(* Logix 5000 project; controller CLASE_1 Emulate 5570 rev 28.11; software revision 28.02; part 11 of 15 *)
(* tags used below, declared in another part *)
   Cfg_FailOpen : BOOL;   // 1=Fail Open (energize to close), 0=Fail Closed (energize to open)
   PCmd_Open : BOOL;   // Program Command to Open Valve
   PCmd_Close : BOOL;   // Program Command to Close Valve
   OCmd_Open : BOOL;   // Operator Command to Open Valve
   OCmd_Close : BOOL;   // Operator Command to Close Valve
   Out : BOOL;   // 1=Energize Valve Solenoid
   P_ValveSO : BOOL;   // Unique Parameter Name for auto - discovery
   Wrk_Open : BOOL;   // 1=Requested to OPEN Valve, 0=Requested to CLOSE Valve
   Wrk_SimOpenT : TIMER;   // Simulation Delay until Opened
   Wrk_SimCloseT : TIMER;   // Simulation Delay until Closed
   Wrk_TransitStallT : TIMER;   // Timer for Transit Stall Check
   Wrk_FullStallT : TIMER;   // Timer for Full Stall Check
   Wrk_SimOpenLS : BOOL;   // Simulated valve Open Limit Switch
   Wrk_SimClosedLS : BOOL;   // Simulated valve Closed Limit Switch
(* P_ValveSO, continued *)

ROUTINE Prescan   (* ladder *)
// Clear Ownership, set to De-Energized state, clear "lurking" Commands
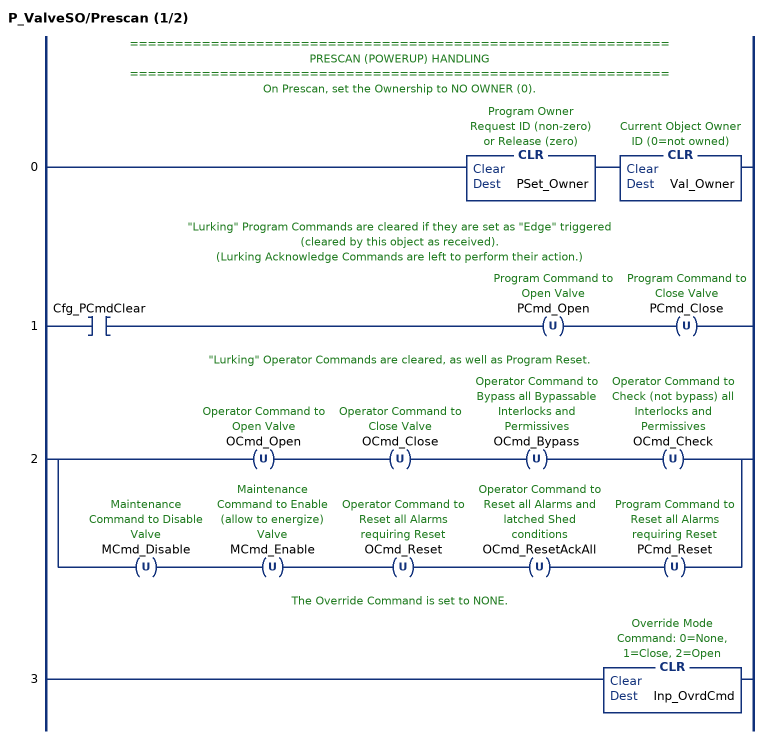
   // ============================================================
   // PRESCAN (POWERUP) HANDLING
   // ============================================================
   // On Prescan, set the Ownership to NO OWNER (0).
   0: CLR(PSet_Owner)CLR(Val_Owner);
   // "Lurking" Program Commands are cleared if they are set as "Edge" triggered
   // (cleared by this object as received).
   // (Lurking Acknowledge Commands are left to perform their action.)
   1: XIC(Cfg_PCmdClear)OTU(PCmd_Open)OTU(PCmd_Close);
   // "Lurking" Operator Commands are cleared, as well as Program Reset.
   2: [OTU(OCmd_Open) OTU(OCmd_Close) OTU(OCmd_Bypass) OTU(OCmd_Check) ,OTU(MCmd_Disable) OTU(MCmd_Enable) OTU(OCmd_Reset) OTU(OCmd_ResetAckAll) OTU(PCmd_Reset) ];
   // The Override Command is set to NONE.
   3: CLR(Inp_OvrdCmd);
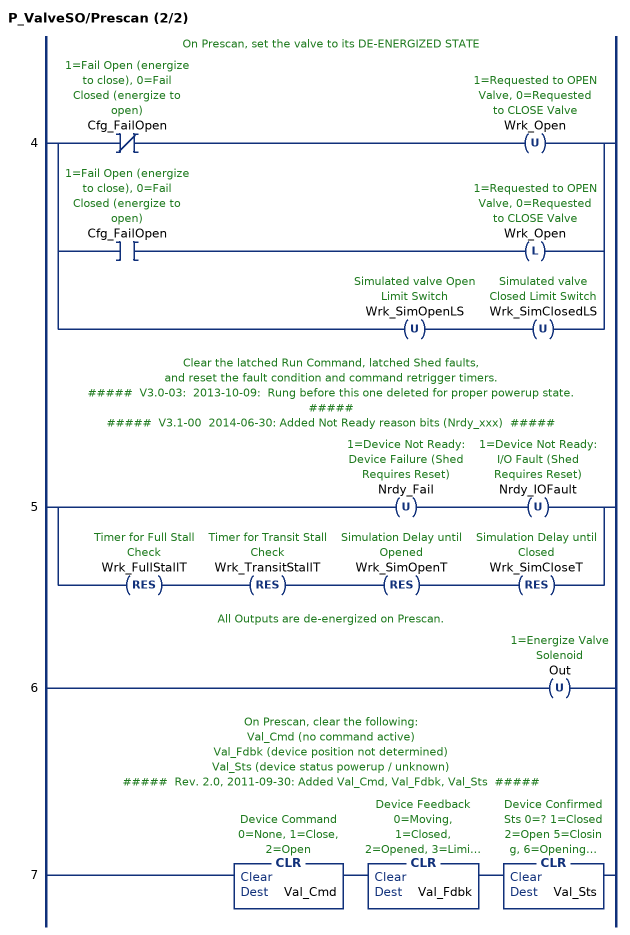
   // On Prescan, set the valve to its DE-ENERGIZED STATE
   4: [XIO(Cfg_FailOpen) OTU(Wrk_Open) ,XIC(Cfg_FailOpen) OTL(Wrk_Open) ,OTU(Wrk_SimOpenLS) OTU(Wrk_SimClosedLS) ];
   // Clear the latched Run Command, latched Shed faults,
   // and reset the fault condition and command retrigger timers.
   // #####  V3.0-03:  2013-10-09:  Rung before this one deleted for proper powerup state.  #####
   // #####  V3.1-00  2014-06-30: Added Not Ready reason bits (Nrdy_xxx)  #####
   5: [OTU(Nrdy_Fail) OTU(Nrdy_IOFault) ,RES(Wrk_FullStallT) RES(Wrk_TransitStallT) RES(Wrk_SimOpenT) RES(Wrk_SimCloseT) ];
   // All Outputs are de-energized on Prescan.
   6: OTU(Out);
   // On Prescan, clear the following:
   // Val_Cmd (no command active)
   // Val_Fdbk (device position not determined)
   // Val_Sts (device status powerup / unknown)
   // #####  Rev. 2.0, 2011-09-30: Added Val_Cmd, Val_Fdbk, Val_Sts  #####
   7: CLR(Val_Cmd)CLR(Val_Fdbk)CLR(Val_Sts);
END_ROUTINE
END_ADD_ON_INSTRUCTION

ADD_ON_INSTRUCTION P_VSD   (* revision 3.5 09 Release, vendor Rockwell Automation, ExecutePrescan, ExecuteEnableInFalse *)
// Variable Speed Drive
// Revision note:
// See V3.5-xx Release Notes for details. Modified to correct indication of motor RUNNING status in HAND mode, regardless of interlock/stop conditions.
// Help:
// Copyright © Rockwell Automation, Inc.  All Rights Reserved.
// This Instruction controls and monitors a Variable-Speed (AC or DC) Drive
// and provides:
// *  Starting drive, stopping drive, jogging drive, setting speed reference and setting direction
// *  Monitoring of run feedback, display of actual drive status, including accel, decel, direction, speed
// *  Detection of Failure to Start, Failure to Stop, Drive Fault/Not Ready
// *  Monitoring of Permissive conditions to allow starting
// *  Monitoring of Interlock conditions to stop drive or prevent starting
// *  Simulation, providing feedback of a working drive while disabling outputs
// *  Monitoring of I/O communication faults
// *  Alarms for Fail to Start, Fail to Stop, Interlock Trip, Drive Fault/Not Ready, I/O Fault
// *  Operation in Hand, Maintenance, Override, Program and Operator Modes
// *  "Available" status for use by automation logic to know whether drive
//       can be controlled by other objects.
// Modes are provided by a P_Mode AOI instance.
// Alarms are provided by P_Alarm AOI instances.
// Modes of operation: Operator, Program, Override, Maintenance, Hand
VAR_IN_OUT
   Ref_FaultCodeList : P_DescList[1]; {required}   // Tag containing List of Fault Codes (DINT) and their Descriptions (STRING)
END_VAR
VAR_INPUT
   Inp_SpeedFdbk : REAL; {visible}   // Speed Feedbak in Drive Units (typ. 0-32767 = 0 to max freq.)
   Inp_LastFaultCode : DINT;   // Most recent drive fault code (enumeration)
   Inp_Datalink : REAL; {visible}   // Auxiliary Signal (datalink) Input in Drive (raw) Units
   Inp_Ready : BOOL := 1; {visible}   // 1=Drive is ready to run
   Inp_Running : BOOL; {visible}   // 1=Drive is Running (active)
   Inp_CommandDir : BOOL := 1; {visible}   // 1=Drive is commanded Forward, 0=Drive is commanded Reverse
   Inp_ActualDir : BOOL := 1; {visible}   // 1=Drive is running Forward, 0=Drive is running Reverse
   Inp_Accelerating : BOOL; {visible}   // 1=Drive is accelerating
   Inp_Decelerating : BOOL; {visible}   // 1=Drive is decelerating
   Inp_Alarm : BOOL; {visible}   // 1=Drive has an Alarm Condition (see drive display or manual)
   Inp_Faulted : BOOL; {visible}   // 1=Drive has Faulted (see drive display or manual)
   Inp_AtSpeed : BOOL; {visible}   // 1=Drive is at commanded speed
   Inp_FwdPermOK : BOOL := 1; {visible}   // 1=Permissives OK, drive can start Forward
   Inp_FwdNBPermOK : BOOL := 1; {visible}   // 1=Non-Bypassable Permissives OK, drive can start Forward
   Inp_RevPermOK : BOOL := 1; {visible}   // 1=Permissives OK, drive can start Reverse
   Inp_RevNBPermOK : BOOL := 1; {visible}   // 1=Non-Bypassable Permissives OK, motor can start Reverse
   Inp_IntlkOK : BOOL := 1; {visible}   // 1=Interlocks OK, drive can start/run
   Inp_NBIntlkOK : BOOL := 1; {visible}   // 1=Non-Bypassable Interlocks OK, drive can start/run
   Inp_IOFault : BOOL;   // Input Communication Status 0=OK, 1=fail
   Inp_Sim : BOOL;   // 1=Simulate working drive; 0=Start/Stop/ Monitor actual drive
   Inp_Hand : ALIAS FOR Mode.Inp_Hand; {visible}
   Inp_Ovrd : ALIAS FOR Mode.Inp_Ovrd; {visible}
   Inp_OvrdCmd : SINT; {visible}   // Override Mode Command: 0=None, 1=Stop, 2=Start Fwd 3=Start Rev
   Inp_OvrdSpeed : REAL;   // Value to set Speed Reference in Override Mode (SpeedRef EU)
   Inp_OvrdOutDatalink : REAL;   // Value to set Output Datalink in Override Mode (OutDatalink EU)
   Inp_Reset : BOOL; {visible}   // 1=Reset drive fault conditions and latched Alarms
   Cfg_HasReverse : BOOL;   // 1=Drive can be run reverse, 0=Forward only
   Cfg_HasJog : BOOL;   // 1=Drive Jog Command enabled/visible, 0=Drive Jog Command not allowed
   Cfg_AllowLocal : BOOL;   // 1=Allow Local Start/Stop without alarm, 0=Start/Stop from HMI/prog only
   Cfg_HasRunFdbk : BOOL;   // 1=Drive provides feedback signal on Inp_Running when running
   Cfg_UseRunFdbk : BOOL;   // 1=Drive run feedback should be used for failure checking
   Cfg_HasSpeedFdbk : BOOL;   // 1=Drive provides speed feedback on Inp_SpeedFdbk
   Cfg_UseSpeedFdbk : BOOL;   // 1=Drive speed determines running state, 0=state determined by drive Active input bit
   Cfg_HasInpDatalink : BOOL;   // 1=A signal is connected to Inp_Datalink
   Cfg_HasOutDatalink : BOOL;   // 1=A signal is connected to Out_Datalink
   Cfg_HasFwdPermObj : BOOL;   // 1=Tells HMI a P_Perm is connected to Inp_FwdPerm
   Cfg_HasRevPermObj : BOOL;   // 1=Tells HMI a P_Perm is connected to Inp_RevPerm
   Cfg_HasIntlkObj : BOOL;   // 1=Tells HMI a P_Intlk is connected to Inp_Intlk
   Cfg_HasResInhObj : BOOL;   // 1=Tells HMI a P_ResInh Restart Inhibit is connected
   Cfg_HasRunTimeObj : BOOL;   // 1=Tells HMI a P_RunTime is connected
   Cfg_SetTrack : BOOL := 1;   // 1=PSets track OSets in Oper, OSets track PSets in Prog, 0=no tracking
   Cfg_SetTrackOvrdHand : BOOL;   // 1=Prog/Oper Settings track Override/Hand speed reference
   Cfg_PCmdClear : ALIAS FOR Mode.Cfg_PCmdClear;
   Cfg_ProgDefault : ALIAS FOR Mode.Cfg_ProgDefault;
   Cfg_OperStopPrio : BOOL;   // 1=OCmd_Stop has priority, accepted any time, 0=OCmd_Stop only in Oper, Maint Mode.
   Cfg_OCmdResets : BOOL;   // 1=New Oper drive cmd. resets fault, 0=reset req'd to clear fault
   Cfg_OvrdPermIntlk : BOOL;   // 1=Override ignores Bypassable Perm/ Intlk; 0=always use Perm/Intlk
   Cfg_ShedOnFailToStart : BOOL := 1;   // 1=Stop Motor and Alarm on Fail to Start; 0=Alarm only on Fail to Start
   Cfg_ShedOnIOFault : BOOL := 1;   // 1=Stop Motor and Alarm on I/O Fault; 0=Alarm only on I/O Fault
   Cfg_SimScaleEU : BOOL;   // 1=In simulation, scale Speed Ref EU to Speed Fdbk EU
   Cfg_SimScaleRaw : BOOL;   // 1=In simulation, scale Speed Ref EU to raw, then raw to Speed Fdbk EU
   Cfg_HasFailToStartAlm : ALIAS FOR FailToStart.Cfg_Exists;   // 1=Fail to Start Alarm exists and will be checked
   Cfg_HasFailToStopAlm : ALIAS FOR FailToStop.Cfg_Exists;   // 1=Fail to Stop Alarm exists and will be checked
   Cfg_HasIntlkTripAlm : ALIAS FOR IntlkTrip.Cfg_Exists;   // 1=Interlock Trip Alarm exists and will be checked
   Cfg_HasDriveFaultAlm : ALIAS FOR DriveFault.Cfg_Exists;   // 1=Drive Fault alarm exists and will be checked
   Cfg_HasIOFaultAlm : ALIAS FOR IOFault.Cfg_Exists;   // 1=I/O Fault Alarm exists and will be checked
   Cfg_FailToStartResetReqd : ALIAS FOR FailToStart.Cfg_ResetReqd;   // 1=Reset requied to clear Fail to Start Alarm
   Cfg_FailToStopResetReqd : ALIAS FOR FailToStop.Cfg_ResetReqd;   // 1=Reset required to clear Fail to Stop Alarm
   Cfg_IntlkTripResetReqd : ALIAS FOR IntlkTrip.Cfg_ResetReqd;   // 1=Reset required to clear Interlock Trip Alarm
   Cfg_DriveFaultResetReqd : ALIAS FOR DriveFault.Cfg_ResetReqd;   // 1=Reset required to clear Drive Fault Alarm
   Cfg_IOFaultResetReqd : ALIAS FOR IOFault.Cfg_ResetReqd;   // 1=Reset required to clear I/O Fault Alarm
   Cfg_FailToStartAckReqd : ALIAS FOR FailToStart.Cfg_AckReqd;   // 1=Acknowledge required for Fail to Start Alarm
   Cfg_FailToStopAckReqd : ALIAS FOR FailToStop.Cfg_AckReqd;   // 1=Acknowledge required for Fail to Stop Alarm
   Cfg_IntlkTripAckReqd : ALIAS FOR IntlkTrip.Cfg_AckReqd;   // 1=Acknowledge required for Interlock Trip Alarm
   Cfg_DriveFaultAckReqd : ALIAS FOR DriveFault.Cfg_AckReqd;   // 1=Acknowledge required for Drive Fault Alarm
   Cfg_IOFaultAckReqd : ALIAS FOR IOFault.Cfg_AckReqd;   // 1=Acknowledge required for I/O Fault Alarm
   Cfg_FailToStartSeverity : ALIAS FOR FailToStart.Cfg_Severity;   // Fail To Start Alarm Severity: 1..250=Low, 251..500=Medium, 501..750=High, 751..1000=Urgent
   Cfg_FailToStopSeverity : ALIAS FOR FailToStop.Cfg_Severity;   // Fail To Stop Alarm Severity: 1..250=Low, 251..500=Medium, 501..750=High, 751..1000=Urgent
   Cfg_IntlkTripSeverity : ALIAS FOR IntlkTrip.Cfg_Severity;   // Interlock Trip Alarm Severity: 1..250=Low, 251..500=Medium, 501..750=High, 751..1000=Urgent
   Cfg_DriveFaultSeverity : ALIAS FOR DriveFault.Cfg_Severity;   // Drive Fault Alarm Severity: 1..250=Low, 251..500=Medium, 501..750=High, 751..1000=Urgent
   Cfg_IOFaultSeverity : ALIAS FOR IOFault.Cfg_Severity;   // I/O Fault Alarm Severity: 1..250=Low, 251..500=Medium, 501..750=High, 751..1000=Urgent
   Cfg_MinSpdRef : REAL;   // Minimum Speed Reference in EU (for limiting)
   Cfg_MaxSpdRef : REAL := 60.0;   // Maximum Speed Reference in EU (for limiting)
   Cfg_SpeedRefRawMin : REAL;   // Speed Reference Minimum in Drive (raw) Units (for scaling)
   Cfg_SpeedRefRawMax : REAL := 32767.0;   // Speed Reference Maximum in Drive (raw) Units (for scaling)
   Cfg_SpeedRefEUMin : REAL;   // Speed Reference Minimum in Engineering Units (for scaling)
   Cfg_SpeedRefEUMax : REAL := 130.0;   // Speed Reference Maximum in Engineering Units (for scaling)
   Cfg_SpeedFdbkRawMin : REAL;   // Speed Feedback Minimum in Drive (raw) Units (for scaling)
   Cfg_SpeedFdbkRawMax : REAL := 32767.0;   // Speed Feedback Maximum in Drive (raw) Units (for scaling)
   Cfg_SpeedFdbkEUMin : REAL;   // Speed Feedback Minimum in Engineering Units (for scaling)
   Cfg_SpeedFdbkEUMax : REAL := 130.0;   // Speed Feedback Maximum in Engineering Units (for scaling)
   Cfg_InpDatalinkRawMin : REAL;   // Input Datalink Minimum in Drive (raw) Units (for scaling)
   Cfg_InpDatalinkRawMax : REAL := 4095.0;   // Input Datalink Maximum in Drive (raw) Units (for scaling)
   Cfg_InpDatalinkEUMin : REAL;   // Input Datalink Minimum in Engineering Units (for scaling)
   Cfg_InpDatalinkEUMax : REAL := 409.5;   // Input Datalink Maximum in Engineering Units (for scaling)
   Cfg_OutDatalinkMin : REAL;   // Minimum Output Datalink in EU (for limiting)
   Cfg_OutDatalinkMax : REAL := 100.0;   // Maximum Output Datalink in EU (for limiting)
   Cfg_OutDatalinkRawMin : REAL;   // Output Datalink Minimum in Drive (raw) Units (for scaling)
   Cfg_OutDatalinkRawMax : REAL := 4095.0;   // Output Datalink Maximum in Drive (raw) Units (for scaling)
   Cfg_OutDatalinkEUMin : REAL;   // Output Datalink Minimum in Engineering Units (for scaling)
   Cfg_OutDatalinkEUMax : REAL := 409.5;   // Output Datalink Maximum in Engineering Units (for scaling)
   Cfg_SimRampT : DINT := 10;   // Time to ramp speed fdbk when in Simulation (sec)
   Cfg_FailToStartT : DINT := 15;   // Time after Start to get Run Feedback before Fault (sec)
   Cfg_FailToStopT : DINT := 15;   // Time after Stop to drop Run Feedback before Fault (sec)
   Cfg_ResetPulseT : DINT := 2;   // Time to pulse Out_Reset to clear drive fault
   Cfg_MaxJogT : REAL;   // Maximum jog time (sec, 0=unlimited)
   Cfg_OperKeep : SINT;   // Oper keeps control in Prog Mode: .0=Reference, .1=Start/Stop, .2=Fwd/Rev, .3=OutDatalink
   Cfg_ProgKeep : SINT;   // Prog keeps control in Oper Mode: .0=Reference, .1=Start/Stop, .2=Fwd/Rev, .3=OutDatalink
   PSet_SpeedRef : REAL;   // Program Setting of Speed Reference (EU)
   PSet_OutDatalink : REAL;   // Program Setting of Output Datalink (EU)
   PSet_Owner : DINT;   // Program Owner Request ID (non-zero) or Release (zero)
   OSet_SpeedRef : REAL;   // Operator Setting of Speed Reference (EU)
   OSet_OutDatalink : REAL;   // Operator Setting of Output Datalink (EU)
   PCmd_Start : BOOL;   // Program Command to Start Drive
   PCmd_Stop : BOOL;   // Program Command to Stop Drive
   PCmd_Fwd : BOOL;   // Program Command to set direction to Fowrard
   PCmd_Rev : BOOL;   // Program Command to set direction to Reverse
   PCmd_Acq : ALIAS FOR Mode.PCmd_Acq;
   PCmd_Rel : ALIAS FOR Mode.PCmd_Rel;
   PCmd_Lock : ALIAS FOR Mode.PCmd_Lock;
   PCmd_Unlock : ALIAS FOR Mode.PCmd_Unlock;
   PCmd_Reset : BOOL;   // Program Command to Reset drive fault and all Alarms requiring Reset
   PCmd_FailToStartAck : ALIAS FOR FailToStart.PCmd_Ack;   // Program Command to Acknowledge Fail to Start Alarm
   PCmd_FailToStartSuppress : ALIAS FOR FailToStart.PCmd_Suppress;   // Program Command to Suppress Fail to Start Alarm
   PCmd_FailToStartUnsuppress : ALIAS FOR FailToStart.PCmd_Unsuppress;   // Program Command to Unsuppress Fail to Start Alarm
   PCmd_FailToStartUnshelve : ALIAS FOR FailToStart.PCmd_Unshelve;   // Program Command to Unshelve Fail to Start Alarm
   PCmd_FailToStopAck : ALIAS FOR FailToStop.PCmd_Ack;   // Program Command to Acknowledge Fail to Stop Alarm
   PCmd_FailToStopSuppress : ALIAS FOR FailToStop.PCmd_Suppress;   // Program Command to Suppress Fail to Stop Alarm
   PCmd_FailToStopUnsuppress : ALIAS FOR FailToStop.PCmd_Unsuppress;   // Program Command to Unsuppress Fail to Stop Alarm
   PCmd_FailToStopUnshelve : ALIAS FOR FailToStop.PCmd_Unshelve;   // Program Command to Unshelve Fail to Stop Alarm
   PCmd_IntlkTripAck : ALIAS FOR IntlkTrip.PCmd_Ack;   // Program Command to Acknowledge Interlock Trip Alarm
   PCmd_IntlkTripSuppress : ALIAS FOR IntlkTrip.PCmd_Suppress;   // Program Command to Suppress Interlock Trip Alarm
   PCmd_IntlkTripUnsuppress : ALIAS FOR IntlkTrip.PCmd_Unsuppress;   // Program Command to Unsuppress Interlock Trip Alarm
   PCmd_IntlkTripUnshelve : ALIAS FOR IntlkTrip.PCmd_Unshelve;   // Program Command to Unshelve Interlock Trip Alarm
   PCmd_DriveFaultAck : ALIAS FOR DriveFault.PCmd_Ack;   // Program Command to Acknowledge Drive Fault Alarm
   PCmd_DriveFaultSuppress : ALIAS FOR DriveFault.PCmd_Suppress;   // Program Command to Suppress Drive Fault Alarm
   PCmd_DriveFaultUnsuppress : ALIAS FOR DriveFault.PCmd_Unsuppress;   // Program Command to Unsuppress Drive Fault Alarm
   PCmd_DriveFaultUnshelve : ALIAS FOR DriveFault.PCmd_Unshelve;   // Program Command to Unshelve Drive Fault Alarm
   PCmd_IOFaultAck : ALIAS FOR IOFault.PCmd_Ack;   // Program Command to Acknowledge I/O Fault Alarm
   PCmd_IOFaultSuppress : ALIAS FOR IOFault.PCmd_Suppress;   // Program Command to Suppress I/O Fault Alarm
   PCmd_IOFaultUnsuppress : ALIAS FOR IOFault.PCmd_Unsuppress;   // Program Command to Unsuppress I/O Fault Alarm
   PCmd_IOFaultUnshelve : ALIAS FOR IOFault.PCmd_Unshelve;   // Program Command to Unshelve I/O Fault Alarm
   OCmd_Start : BOOL;   // Operator Command to Start Drive
   OCmd_Stop : BOOL;   // Operator Command to Stop Drive
   OCmd_Jog : BOOL;   // Operator Command to Jog Drive (not cleared by P_VSD!)
   OCmd_Fwd : BOOL;   // Operator Command to set direction to Forward
   OCmd_Rev : BOOL;   // Operator Command to set direction to Reverse
   OCmd_Bypass : BOOL;   // Operator Command to Bypass all Bypassable Interlocks and Permissives
   OCmd_Check : BOOL;   // Operator Command to Check (not bypass) all Interlocks and Permissives
   MCmd_Disable : BOOL;   // Maintenance Command to Disable Drive
   MCmd_Enable : BOOL;   // Maintenance Command to Enable (allow to run) Drive
   MCmd_Acq : ALIAS FOR Mode.MCmd_Acq;
   MCmd_Rel : ALIAS FOR Mode.MCmd_Rel;
   OCmd_AcqLock : ALIAS FOR Mode.OCmd_AcqLock;
   OCmd_Unlock : ALIAS FOR Mode.OCmd_UnlockRel;
   OCmd_Reset : BOOL;   // Operator Command to Reset all Alarms requiring Reset
   OCmd_ResetAckAll : BOOL;   // Operator Command to Reset all Alarms and latched Shed conditions
END_VAR
VAR_OUTPUT
   Out_SpeedRef : REAL; {access Read Only, visible}   // Drive Speed Reference in Drive Units (typ. 0-32767 = 0 to max freq.)
   Out_Datalink : REAL; {access Read Only, visible}   // Auxiliary Signal (datalink) Output in Drive (raw) Units
   Out_Run : BOOL; {access Read Only}   // 1=Start/Run Drive, 0=Stop Drive (for held starter type)
   Out_Stop : BOOL; {access Read Only, visible}   // 1=Stop Drive, 0=drive left in current state
   Out_Start : BOOL; {access Read Only, visible}   // 1=Start Drive, 0=drive left in current state
   Out_Jog : BOOL; {access Read Only, visible}   // 1=Jog drive at Jog Speed, -->0=stop jogging
   Out_ClearFault : BOOL; {access Read Only, visible}   // 1=Attempt to clear Drive Fault
   Out_Fwd : BOOL; {access Read Only, visible}   // 1=Set drive direction to Forward
   Out_Rev : BOOL; {access Read Only, visible}   // 1=Set drive direction to Reverse
   Val_SpeedRef : REAL; {access Read Only, visible}   // Speed Reference (target) to drive
   Val_SpeedFdbk : REAL; {access Read Only, visible}   // Speed Feedback (actual) from drive
   Val_InpDatalink : REAL; {access Read Only, visible}   // Input Datalink value from drive
   Val_OutDatalink : REAL; {access Read Only, visible}   // Output Datalink value to drive
   Val_SpeedRefEUMin : REAL; {access Read Only}   // Minimum of Speed Reference = MIN (Cfg_SpeedFdbkEUMin, Cfg_SpeedFdbkEUMax)
   Val_SpeedRefEUMax : REAL := 130.0; {access Read Only}   // Maximum of Speed Reference = MAX (Cfg_SpeedFdbkEUMin, Cfg_SpeedFdbkEUMax)
   Val_SpeedFdbkEUMin : REAL; {access Read Only}   // Minimum of Speed Feedback = MIN (Cfg_SpeedFdbkEUMin, Cfg_SpeedFdbkEUMax)
   Val_SpeedFdbkEUMax : REAL := 130.0; {access Read Only}   // Maximum of Speed Feedback = MAX (Cfg_SpeedFdbkEUMin, Cfg_SpeedFdbkEUMax)
   Val_LastFaultCode : DINT; {access Read Only}   // Most recent drive fault code (enumeration)
   SrcQ_IO : SINT; {access Read Only}   // Source and Quality of primary I/O (enumeration)
   SrcQ : SINT; {access Read Only}   // Source and Quality of primary Val/Sts (enumeration)
   Val_Cmd : SINT; {access Read Only}   // Device Command 0=None, 1=Stop, 2=StartFwd 3=StartRev 4=JogFwd 5=JogRev
   Val_Fdbk : SINT; {access Read Only}   // Device Feedback 0=Stopped, 1=Running Fwd 2=Running Rev 3=Accelerating 4=Decelerating
   Val_Sts : SINT; {access Read Only}   // Device Confirmed Sts 0? 1=Stop 2=RunF 3=RunR 4=JogF 5=JogR 6=Stopping 7=Starting F 8=Starting R, 33=Disabled
   Val_Fault : SINT; {access Read Only, visible}   // Device Fault Status 0=None, 16=Fail to Start, 17 = Fail to Stop, 18=Drive Fault, 32=I/O Fault, 34=Config Error
   Val_Mode : ALIAS FOR Mode.Val; {access Read Only}
   Val_Owner : DINT; {access Read Only}   // Current Object Owner ID (0=not owned)
   Val_Notify : SINT; {access Read Only}   // Current Alarm Level and Acknowledgement (enumeration)
   Sts_Stopped : BOOL; {access Read Only, visible}   // 1=Drive requested to stop and is confirmed stopped
   Sts_Starting : BOOL; {access Read Only, visible}   // 1=Drive requested to run and awaiting run feedback
   Sts_Running : BOOL; {access Read Only, visible}   // 1=Drive requested to run and is confirmed running
   Sts_Stopping : BOOL; {access Read Only, visible}   // 1=Drive requested to stop and awaiting stopped feedback
   Sts_Jogging : BOOL; {access Read Only, visible}   // 1=Drive requested to Jog
   Sts_CommandDir : BOOL; {access Read Only}   // 1=Drive commanded to Forward, 0=Reverse
   Sts_ActualDir : BOOL; {access Read Only, visible}   // 1=Drive Actual direction is Forward, 0=Reverse
   Sts_Accel : BOOL; {access Read Only}   // 1=Drive is Accelerating
   Sts_Decel : BOOL; {access Read Only}   // 1=Drive is Decelerating
   Sts_NotReady : BOOL; {access Read Only}   // 1=Drive is Not Ready (cannot be started) Check alarms, stops, faults
   Sts_Alarm : BOOL; {access Read Only, visible}   // 1=Drive has an Alarm (see drive display or manual)
   Sts_AtSpeed : BOOL; {access Read Only, visible}   // 1=Drive is running at reference speed
   Sts_SpeedLimited : BOOL; {access Read Only, visible}   // 1=Speed Reference Setting exceeds configured Max/Min limit
   Sts_Available : BOOL; {access Read Only, visible}   // 1=Drive available for control by automation (Prog)
   Sts_Bypass : BOOL; {access Read Only}   // 1=Bypassable Interlocks and Permissives are Bypassed
   Sts_BypActive : BOOL; {access Read Only}   // 1=Bypassing Active (Bypassed or Maintenance)
   Sts_Disabled : BOOL; {access Read Only}   // 1=Drive is Disabled
   Sts_NotRdy : BOOL; {access Read Only}   // 1=Device Not Ready, see detail bits for reason
   Nrdy_Disabled : BOOL; {access Read Only}   // 1=Device Not Ready: Device Disabled by Maintenance
   Nrdy_CfgErr : BOOL; {access Read Only}   // 1=Device Not Ready: Configuration Error
   Nrdy_Intlk : BOOL; {access Read Only}   // 1=Device Not Ready: Interlock Not OK
   Nrdy_Perm : BOOL; {access Read Only}   // 1=Device Not Ready: Permissive Not OK
   Nrdy_OperPrio : BOOL; {access Read Only}   // 1=Device Not Ready: Operator State 0 Priority Command Requires Reset
   Nrdy_Fail : BOOL; {access Read Only}   // 1=Device Not Ready: Device Failure (Shed Requires Reset)
   Nrdy_IOFault : BOOL; {access Read Only}   // 1=Device Not Ready: I/O Fault (Shed Requires Reset)
   Nrdy_Trip : BOOL; {access Read Only}   // 1=Device not Ready: Deivce Tripped (Drive Fault)
   Nrdy_DriveNR : BOOL; {access Read Only}   // 1=Device Note Ready: Drive Not Ready
   Nrdy_NoMode : BOOL; {access Read Only}   // 1=Device Not Ready: Device Logic Disabled / NO Mode
   Sts_MaintByp : BOOL; {access Read Only}   // 1=A Maintenance Bypass is Active, display icon
   Sts_AlmInh : BOOL; {access Read Only}   // 1=An Alarm is Shelved, Disabled or Suppressed, display icon
   Sts_Err : BOOL; {access Read Only, visible}   // 1=Error in Config: see detail bits for reason
   Err_Timer : BOOL; {access Read Only}   // 1=Error in Config: Invalid Check or Reset Pulse Time (use 0 to 2147483)
   Err_Sim : BOOL; {access Read Only}   // 1=Error in Config: simulation timer preset: use 0 to 2147483)
   Err_Alarm : BOOL; {access Read Only}   // 1=Error in Config: Alarm Min On Time, Shelf Time, Severity
   Err_FdbkRaw : BOOL; {access Read Only}   // 1=Erron in Config: Speed Fdbk Raw Min = Max
   Err_FdbkEU : BOOL; {access Read Only}   // 1=Error in Config: Speed Fdbk EU Min = Max
   Err_RefLim : BOOL; {access Read Only}   // 1=Error in Config: Speed Ref Limit Min > Max
   Err_RefEU : BOOL; {access Read Only}   // 1=Error in Config: Speed Ref EU Min = Max
   Err_RefRaw : BOOL; {access Read Only}   // 1=Error in Config: Speed Ref Raw Min = Max
   Err_InpDLRaw : BOOL; {access Read Only}   // 1=Error in Config: Input Datalink Raw Min = Max
   Err_InpDLEU : BOOL; {access Read Only}   // 1=Error in Config: Input Datalink EU Min = Max
   Err_OutDLLim : BOOL; {access Read Only}   // 1=Error in Config: Output Datalink Limits Min > Max
   Err_OutDLEU : BOOL; {access Read Only}   // 1=Error in Config: Output Datalink EU Min = Max
   Err_OutDLRaw : BOOL; {access Read Only}   // 1=Error in Config: Output Datalink Raw Min = Max
   Sts_Hand : ALIAS FOR Mode.Sts_Hand; {access Read Only, visible}
   Sts_Maint : ALIAS FOR Mode.Sts_Maint; {access Read Only, visible}
   Sts_Ovrd : ALIAS FOR Mode.Sts_Ovrd; {access Read Only, visible}
   Sts_Prog : ALIAS FOR Mode.Sts_Prog; {access Read Only, visible}
   Sts_Oper : ALIAS FOR Mode.Sts_Oper; {access Read Only, visible}
   Sts_ProgOperLock : ALIAS FOR Mode.Sts_ProgOperLock; {access Read Only}
   Sts_NoMode : ALIAS FOR Mode.Sts_NoMode; {access Read Only}
   Sts_MAcqRcvd : ALIAS FOR Mode.Sts_MAcqRcvd; {access Read Only}
   Sts_FailToStart : ALIAS FOR FailToStart.Inp;   // 1=Drive Failed to Start (One-Shot)
   Alm_FailToStart : ALIAS FOR FailToStart.Alm;   // 1=Drive Fail to Start Alarm
   Ack_FailToStart : ALIAS FOR FailToStart.Ack;   // 1=Fail to Start Alarm has been acknowledged
   Sts_FailToStartDisabled : ALIAS FOR FailToStart.Disabled;   // 1=Fail to Start Alarm has been Disabled by Maintenance
   Sts_FailToStartShelved : ALIAS FOR FailToStart.Shelved;   // 1=Fail to Start Alarm has been Shelved by Operator
   Sts_FailToStartSuppressed : ALIAS FOR FailToStart.Suppressed;   // 1=Fail to Start Alarm has been Suppressed by Program
   Sts_FailToStop : ALIAS FOR FailToStop.Inp;   // 1=Drive Failed to Stop
   Alm_FailToStop : ALIAS FOR FailToStop.Alm;   // 1=Drive Fail to Stop Alarm
   Ack_FailToStop : ALIAS FOR FailToStop.Ack;   // 1=Fail to Stop Alarm has been acknowledged
   Sts_FailToStopDisabled : ALIAS FOR FailToStop.Disabled;   // 1=Fail to Stop Alarm has been Disabled by Maintenance
   Sts_FailToStopShelved : ALIAS FOR FailToStop.Shelved;   // 1=Fail to Stop Alarm has been Shelved by Operator
   Sts_FailToStopSuppressed : ALIAS FOR FailToStop.Suppressed;   // 1=Fail to Stop Alarm has been Suppressed by Program
   Sts_IntlkTrip : ALIAS FOR IntlkTrip.Inp;   // 1=Drive was stopped by an Interlock NOT OK (One-Shot)
   Alm_IntlkTrip : ALIAS FOR IntlkTrip.Alm;   // 1=Alarm: Drive stopped by an Interlock NOT OK
   Ack_IntlkTrip : ALIAS FOR IntlkTrip.Ack;   // 1=Interlock Trip Alarm has been acknowledged
   Sts_IntlkTripDisabled : ALIAS FOR IntlkTrip.Disabled;   // 1=Interlock Trip Alarm has been Disabled by Maintenance
   Sts_IntlkTripShelved : ALIAS FOR IntlkTrip.Shelved;   // 1=Interlock Trip Alarm has been Shelved by Operator
   Sts_IntlkTripSuppressed : ALIAS FOR IntlkTrip.Suppressed;   // 1=Interlock Trip Alarm has been Suppressed by Program
   Sts_DriveFault : ALIAS FOR DriveFault.Inp;   // 1=Drive Fault (see drive display or manual)
   Alm_DriveFault : ALIAS FOR DriveFault.Alm;   // 1=Alarm: Drive Fault (see drive display or manual)
   Ack_DriveFault : ALIAS FOR DriveFault.Ack;   // 1=Drive Fault Alarm has been acknowledged
   Sts_DriveFaultDisabled : ALIAS FOR DriveFault.Disabled;   // 1=Drive Fault Alarm has been Disabled by Maintenance
   Sts_DriveFaultShelved : ALIAS FOR DriveFault.Shelved;   // 1=Drive Fault Alarm has been Shelved by Operator
   Sts_DriveFaultSuppressed : ALIAS FOR DriveFault.Suppressed;   // 1=Drive Fault Alarm has been Suppressed by Program
   Sts_IOFault : ALIAS FOR IOFault.Inp;   // I/O Comm Fault Status (0=OK, 1=Bad)
   Alm_IOFault : ALIAS FOR IOFault.Alm;   // 1=I/O Fault Alarm
   Ack_IOFault : ALIAS FOR IOFault.Ack;   // 1=I/O Fault Alarm has been acknowledged
   Sts_IOFaultDisabled : ALIAS FOR IOFault.Disabled;   // 1=I/O Fault Alarm has been Disabled by Maintenance
   Sts_IOFaultShelved : ALIAS FOR IOFault.Shelved;   // 1=I/O Fault Alarm has been Shelved by Operator
   Sts_IOFaultSuppressed : ALIAS FOR IOFault.Suppressed;   // 1=I/O Fault Alarm has been Suppressed by Program
   Rdy_Start : BOOL; {access Read Only}   // 1=Ready to receive OCmd_Start (enables HMI button)
   Rdy_Stop : BOOL; {access Read Only}   // 1=Ready to receive OCmd_Stop (enables HMI button)
   Rdy_Jog : BOOL; {access Read Only}   // 1=Ready to receive OCmd_Jog (enables HMI button)
   Rdy_Fwd : BOOL; {access Read Only}   // 1=Ready to receive OCmd_Fwd (enabled HMI button)
   Rdy_Rev : BOOL; {access Read Only}   // 1=Ready to receive OCmd_Rev (enables HMI button)
   Rdy_Bypass : BOOL; {access Read Only}   // 1=Ready to receive OCmd_Bypass (enables HMI button)
   Rdy_Check : BOOL; {access Read Only}   // 1=Ready to receive OCmd_Check (enables HMI button)
   Rdy_Disable : BOOL; {access Read Only}   // 1=Ready to receive MCmd_Disable (enables HMI button)
   Rdy_Enable : BOOL; {access Read Only}   // 1=Ready to receive MCmd_Enable (enables HMI button)
   Rdy_Reset : BOOL; {access Read Only}   // 1=Ready to receive OCmd_Reset (enables HMI button)
   Rdy_ResetAckAll : BOOL; {access Read Only}   // 1=At least one Alarm or latched Shed condition requires Reset or Ack
   Rdy_SpeedRef : BOOL; {access Read Only}   // 1=Ready to receive OSet_SpeedRef (enables data entry field)
   Rdy_OSet : BOOL; {access Read Only}   // 1=Ready to receive OSets (other than CV) (enables data entry fields)
   P_VSD : BOOL;   // Unique Parameter Name for auto - discovery
END_VAR
VAR
   Mode : P_Mode := (Cfg_PCmdClear := 1, Cfg_OvrdOverLock := 1, Rdy_OAcq := 1);   // Drive Mode Selection
   IOFault : P_Alarm := (Cfg_AckReqd := 1, Cfg_AllowShelve := 1, Cfg_AllowDisable := 1, Cfg_PCmdClear := 1, Cfg_Severity := 1000, Cfg_AlmMinOnT := 5, PCfg_AllowExist := 1, Ack := 1);   // I/O Fault Alarm
   IntlkTrip : P_Alarm := (Cfg_AckReqd := 1, Cfg_AllowShelve := 1, Cfg_AllowDisable := 1, Cfg_PCmdClear := 1, Cfg_Severity := 500, Cfg_AlmMinOnT := 5, PCfg_AllowExist := 1, Ack := 1);   // Interlock Trip Alarm
   FailToStop : P_Alarm := (Cfg_AckReqd := 1, Cfg_AllowShelve := 1, Cfg_AllowDisable := 1, Cfg_PCmdClear := 1, Cfg_Severity := 1000, Cfg_AlmMinOnT := 5, PCfg_AllowExist := 1, Ack := 1);   // Drive Failed to Stop Alarm
   FailToStart : P_Alarm := (Cfg_AckReqd := 1, Cfg_AllowShelve := 1, Cfg_AllowDisable := 1, Cfg_PCmdClear := 1, Cfg_Severity := 1000, Cfg_AlmMinOnT := 5, PCfg_AllowExist := 1, Ack := 1);   // Drive Failed to Start Alarm
   Cfg_Tag : STRING_20 := 'P_VSD';   // Tagname for display on HMI
   Cfg_Label : STRING_20 := 'Motor Speed Control';   // Label for graphic symbol displayed on HMI
   Cfg_Desc : STRING_40 := 'Variable Speed Drive';   // Description for display on HMI
   Wrk_Run : BOOL; {access None}   // 1=Drive should be "running", 0=should be "stopped"
   Wrk_StartRetrigT : TIMER; {access None}   // Time to pulse start output on start command retrigger (Maint)
   Wrk_StopRetrigT : TIMER; {access None}   // Time to pulse stop output on stop command retrigger (Maint)
   Wrk_RunFdbk : BOOL; {access None}   // Run Feedback based on mode, simulation, etc. 1=running
   Wrk_Notify : DINT; {access None}   // Buffer for building Val_Notify
   Wrk_Bypass : BOOL; {access None}   // Internal Bypassable Permissives and Interlocks are Bypassed flag
   Wrk_Disabled : BOOL; {access None}   // Internal Drive is Disabled
   DriveFault : P_Alarm := (Cfg_AckReqd := 1, Cfg_AllowShelve := 1, Cfg_AllowDisable := 1, Cfg_PCmdClear := 1, Cfg_Severity := 1000, Cfg_AlmMinOnT := 5, PCfg_AllowExist := 1, Ack := 1);   // Drive Faulted Alarm
   Cfg_SpeedRefEU : STRING_8 := 'Hz';   // Speed Reference Engineering Units for display on HMI
   Wrk_SpeedRef : REAL; {access None}   // Working copy of Speed Reference (for limiting)
   Wrk_Rev : BOOL; {access None}   // Working (internal) Direction 1=Reverse 0=Forward (default)
   Wrk_Jog : BOOL; {access None}   // 1=Jog Drive, 0=Drive not jogging
   Wrk_ResetT : TIMER; {access None}   // Reset Output Pulse Timer
   Wrk_ResetONS : BOOL; {access None}   // One-Shot to fire Reset Timer to ensure min. output ON time.
   Cfg_SpeedFdbkEU : STRING_8 := 'Hz';   // Speed Feedback Engineering Units for display on HMI
   Cfg_OutDatalinkLabel : STRING_20;   // Datalink Output Label displayed on faceplate
   Cfg_InpDatalinkLabel : STRING_20;   // Datalink Input Label displayed on faceplate
   Cfg_OutDatalinkEU : STRING_8;   // Datalink Output Engineering Units for display on HMI
   Cfg_InpDatalinkEU : STRING_8;   // Datalink Input Engineering Units for display on HMI
   Wrk_OutDatalink : REAL; {access None}   // Selected Output Datalink setting
   Cfg_RevText : STRING_16 := 'Reverse';   // Name for Reverse Direction, e.g., "Down", "Reverse"
   Cfg_FwdText : STRING_16 := 'Forward';   // Name for Forward Direction, e.g., "Up", "Forward"
   Wrk_StopT : TIMER; {access Read Only}   // Stop Check Timer (for Fail to Stop)
   Wrk_StartT : TIMER; {access Read Only}   // Start Check Timer (for Fail to Start)
   Inf_Tab : SINT;   // Tab to display (FTView ME)
   Wrk_Cmd : SINT; {access None}   // Buffer for building Val_Cmd
   Wrk_Sts : SINT; {access None}   // Buffer for building Val_Sts
   Wrk_Fault : SINT; {access None}   // Buffer for building Val_Fault
   Wrk_Retrigger : BOOL; {access None}   // Maint Start issued while running or Stop while stopped
   Wrk_Step : REAL; {access None}   // Amount to change simulated Speed Fdbk this scan (ramp)
   Wrk_ScanTime : REAL; {access None}   // Seconds since previous scan
   Wrk_ScanT : TIMER := (PRE := 2147483647); {access None}   // Scan Timer (milliseconds, always runs)
   Wrk_SimFdbkTgt : REAL; {access None}   // Speed Ref converted to Speed Fdbk units for simulation: target speed fdbk
   Inf_Type : STRING_16 := 'P_VSD'; {access Read Only}   // Type identifier for HMI navigation
   Wrk_JogT : TIMER; {access Read Only}   // Jog Timer
   Wrk_FaultDescFSC : CONTROL := (LEN := 1); {access None}   // FSC control for Fault Code List search
   Val_FaultDesc : STRING_40; {access Read Only}   // Description of Drive Fault (given LastFaultCode)
   Wrk_OperKeep3ONS : BOOL; {access None}   // Oper Keep bit 3 one-shot store
   Wrk_OperKeep2ONS : BOOL; {access None}   // Oper Keep bit 2 one-shot store
   Wrk_OperKeep1ONS : BOOL; {access None}   // Oper Keep bit 1 one-shot store
   Wrk_OperKeep0ONS : BOOL; {access None}   // Oper Keep bit 0 one-shot store
   Wrk_ProgKeep3ONS : BOOL; {access None}   // Prog Keep bit 3 one-shot store
   Wrk_ProgKeep2ONS : BOOL; {access None}   // Prog Keep bit 2 one-shot store
   Wrk_ProgKeep1ONS : BOOL; {access None}   // Prog Keep bit 1 one-shot store
   Wrk_ProgKeep0ONS : BOOL; {access None}   // Prog Keep bit 0 one-shot store
   Inf_Lib : STRING_12 := 'RA-BAS'; {access Read Only}   // Display Library for Faceplate call-up
   Wrk_SimScaleEUONS : BOOL; {access None}   // Cfg_SimScaleEU became true this scan
   Wrk_SimScaleRawONS : BOOL; {access None}   // Cfg_SimScaleRaw became true this scan
   Wrk_SrcQ : SINT; {access None}   // Register for building Source / Quality enumeration
   Wrk_NotRdyONS : BOOL; {access None}   // Assert Stop on One-Shot of Sts_NotRdy
   Wrk_NotRdy : BOOL; {access None}   // Device Not Ready conditions excluding shed latches
   Wrk_StartInhT : TIMER; {access None}   // Local Start Inhibit Timer
   Wrk_StopInhT : TIMER; {access None}   // Local Stop Inhibit Timer
   Wrk_NoLongerSim : BOOL; {access None}   // Switched from Simulated to Real Drive this scan
   Wrk_Hand : BOOL; {access None}   // Perform Hand Mode alignment with actual device state
   Wrk_RevCmdRcvd : BOOL; {access None}   // A Reverse direction command was received this scan.
   Wrk_FwdCmdRcvd : BOOL; {access None}   // A Forward direction command was received this scan
END_VAR

ROUTINE EnableInFalse   (* ladder *)
// Disabled is asserted; Outputs OFF; Run Status shown but Alarms disabled
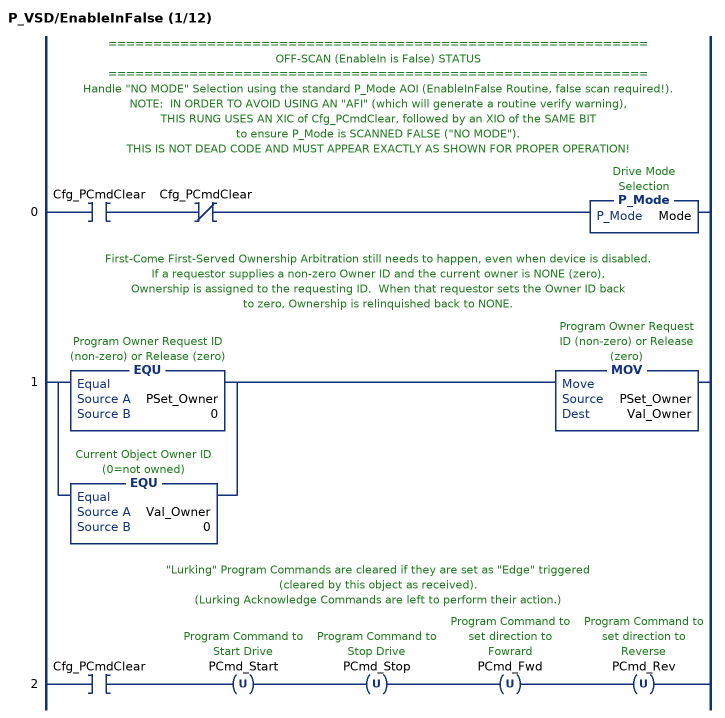
   // ============================================================
   // OFF-SCAN (EnableIn is False) STATUS
   // ============================================================
   // Handle "NO MODE" Selection using the standard P_Mode AOI (EnableInFalse Routine, false scan required!).
   // NOTE:  IN ORDER TO AVOID USING AN "AFI" (which will generate a routine verify warning),
   // THIS RUNG USES AN XIC of Cfg_PCmdClear, followed by an XIO of the SAME BIT
   // to ensure P_Mode is SCANNED FALSE ("NO MODE").
   // THIS IS NOT DEAD CODE AND MUST APPEAR EXACTLY AS SHOWN FOR PROPER OPERATION!
   0: XIC(Cfg_PCmdClear)XIO(Cfg_PCmdClear)P_Mode(Mode);
   // First-Come First-Served Ownership Arbitration still needs to happen, even when device is disabled.
   // If a requestor supplies a non-zero Owner ID and the current owner is NONE (zero),
   // Ownership is assigned to the requesting ID.  When that requestor sets the Owner ID back
   // to zero, Ownership is relinquished back to NONE.
   1: [EQU(PSet_Owner,0) ,EQU(Val_Owner,0) ]MOV(PSet_Owner,Val_Owner);
   // "Lurking" Program Commands are cleared if they are set as "Edge" triggered
   // (cleared by this object as received).
   // (Lurking Acknowledge Commands are left to perform their action.)
   2: XIC(Cfg_PCmdClear)OTU(PCmd_Start)OTU(PCmd_Stop)OTU(PCmd_Fwd)OTU(PCmd_Rev);
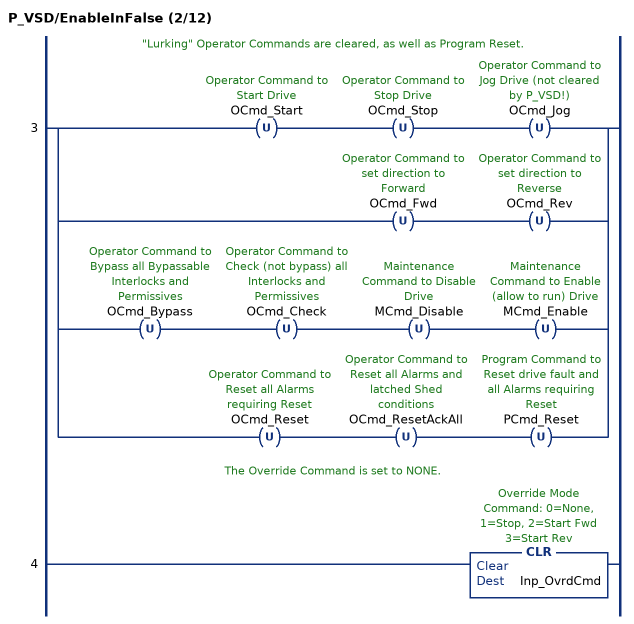
   // "Lurking" Operator Commands are cleared, as well as Program Reset.
   3: [OTU(OCmd_Start) OTU(OCmd_Stop) OTU(OCmd_Jog) ,OTU(OCmd_Fwd) OTU(OCmd_Rev) ,OTU(OCmd_Bypass) OTU(OCmd_Check) OTU(MCmd_Disable) OTU(MCmd_Enable) ,OTU(OCmd_Reset) OTU(OCmd_ResetAckAll) OTU(PCmd_Reset) ];
   // The Override Command is set to NONE.
   4: CLR(Inp_OvrdCmd);
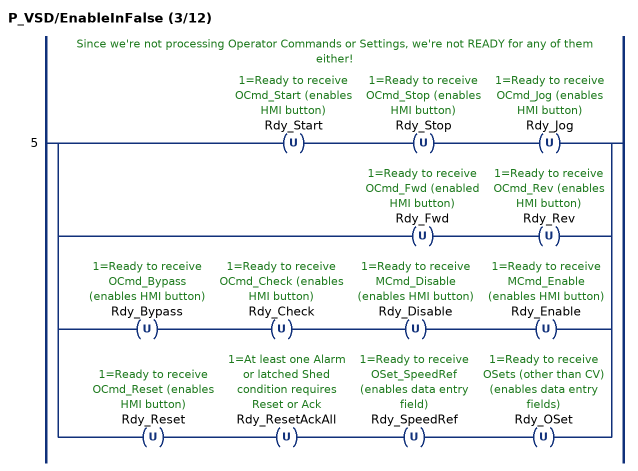
   // Since we're not processing Operator Commands or Settings, we're not READY for any of them either!
   5: [OTU(Rdy_Start) OTU(Rdy_Stop) OTU(Rdy_Jog) ,OTU(Rdy_Fwd) OTU(Rdy_Rev) ,OTU(Rdy_Bypass) OTU(Rdy_Check) OTU(Rdy_Disable) OTU(Rdy_Enable) ,OTU(Rdy_Reset) OTU(Rdy_ResetAckAll) OTU(Rdy_SpeedRef) OTU(Rdy_OSet) ];
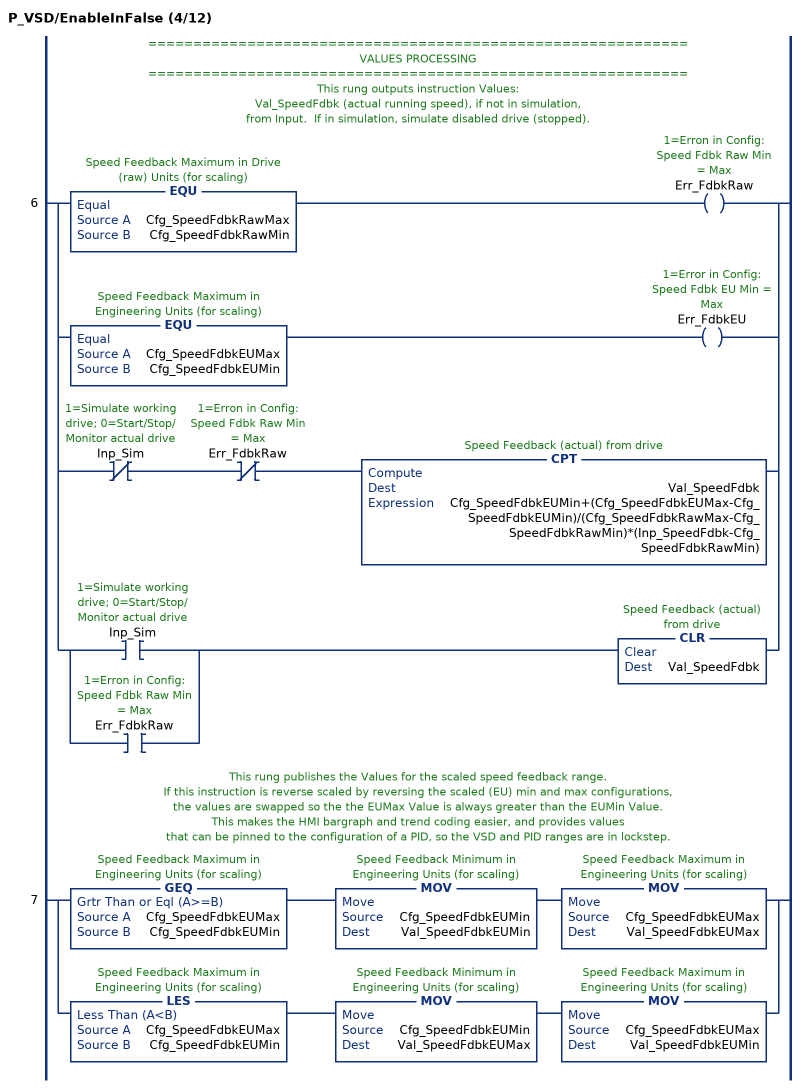
   // ============================================================
   // VALUES PROCESSING
   // ============================================================
   // This rung outputs instruction Values:
   // Val_SpeedFdbk (actual running speed), if not in simulation,
   // from Input.  If in simulation, simulate disabled drive (stopped).
   6: [[EQU(Cfg_SpeedFdbkRawMax,Cfg_SpeedFdbkRawMin) OTE(Err_FdbkRaw) ,EQU(Cfg_SpeedFdbkEUMax,Cfg_SpeedFdbkEUMin) OTE(Err_FdbkEU) ] ,XIO(Inp_Sim) XIO(Err_FdbkRaw) CPT(Val_SpeedFdbk,Cfg_SpeedFdbkEUMin+(Cfg_SpeedFdbkEUMax-Cfg_SpeedFdbkEUMin)/(Cfg_SpeedFdbkRawMax-Cfg_SpeedFdbkRawMin)*(Inp_SpeedFdbk-Cfg_SpeedFdbkRawMin)) ,[XIC(Inp_Sim) ,XIC(Err_FdbkRaw) ] CLR(Val_SpeedFdbk) ];
   // This rung publishes the Values for the scaled speed feedback range.
   // If this instruction is reverse scaled by reversing the scaled (EU) min and max configurations,
   // the values are swapped so the the EUMax Value is always greater than the EUMin Value.
   // This makes the HMI bargraph and trend coding easier, and provides values
   // that can be pinned to the configuration of a PID, so the VSD and PID ranges are in lockstep.
   7: [GEQ(Cfg_SpeedFdbkEUMax,Cfg_SpeedFdbkEUMin) MOV(Cfg_SpeedFdbkEUMin,Val_SpeedFdbkEUMin) MOV(Cfg_SpeedFdbkEUMax,Val_SpeedFdbkEUMax) ,LES(Cfg_SpeedFdbkEUMax,Cfg_SpeedFdbkEUMin) MOV(Cfg_SpeedFdbkEUMin,Val_SpeedFdbkEUMax) MOV(Cfg_SpeedFdbkEUMax,Val_SpeedFdbkEUMin) ];
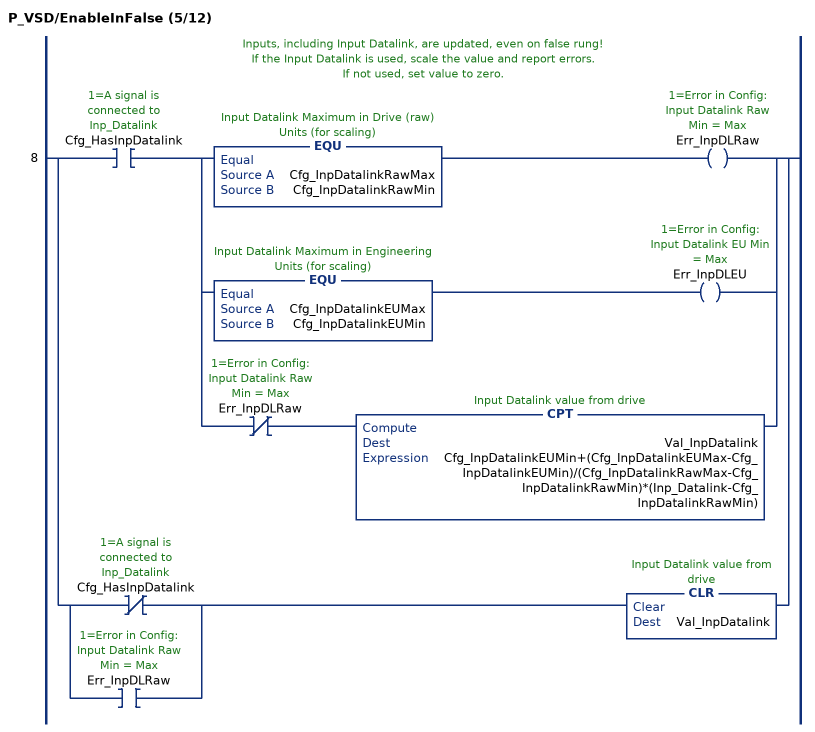
   // Inputs, including Input Datalink, are updated, even on false rung!
   // If the Input Datalink is used, scale the value and report errors.
   // If not used, set value to zero.
   8: [XIC(Cfg_HasInpDatalink) [[EQU(Cfg_InpDatalinkRawMax,Cfg_InpDatalinkRawMin) OTE(Err_InpDLRaw) ,EQU(Cfg_InpDatalinkEUMax,Cfg_InpDatalinkEUMin) OTE(Err_InpDLEU) ] ,XIO(Err_InpDLRaw) CPT(Val_InpDatalink,Cfg_InpDatalinkEUMin+(Cfg_InpDatalinkEUMax-Cfg_InpDatalinkEUMin)/(Cfg_InpDatalinkRawMax-Cfg_InpDatalinkRawMin)*(Inp_Datalink-Cfg_InpDatalinkRawMin)) ] ,[XIO(Cfg_HasInpDatalink) ,XIC(Err_InpDLRaw) ] CLR(Val_InpDatalink) ];
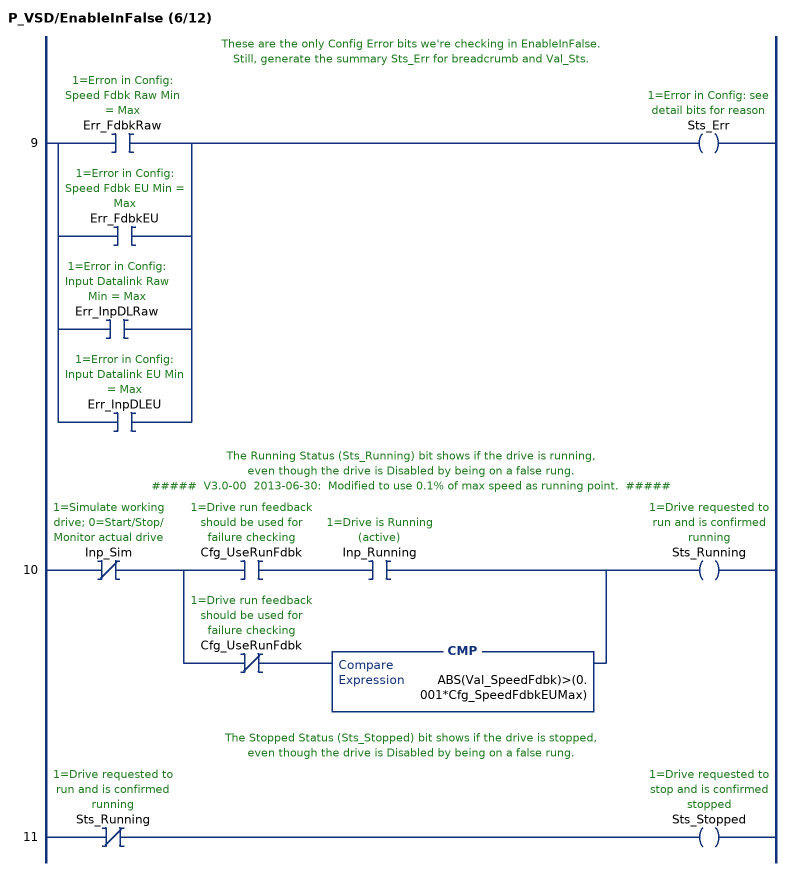
   // These are the only Config Error bits we're checking in EnableInFalse.
   // Still, generate the summary Sts_Err for breadcrumb and Val_Sts.
   9: [XIC(Err_FdbkRaw) ,XIC(Err_FdbkEU) ,XIC(Err_InpDLRaw) ,XIC(Err_InpDLEU) ]OTE(Sts_Err);
   // The Running Status (Sts_Running) bit shows if the drive is running,
   // even though the drive is Disabled by being on a false rung.
   // #####  V3.0-00  2013-06-30:  Modified to use 0.1% of max speed as running point.  #####
   10: XIO(Inp_Sim)[XIC(Cfg_UseRunFdbk) XIC(Inp_Running) ,XIO(Cfg_UseRunFdbk) CMP(ABS(Val_SpeedFdbk)>(0.001*Cfg_SpeedFdbkEUMax)) ]OTE(Sts_Running);
   // The Stopped Status (Sts_Stopped) bit shows if the drive is stopped,
   // even though the drive is Disabled by being on a false rung.
   11: XIO(Sts_Running)OTE(Sts_Stopped);
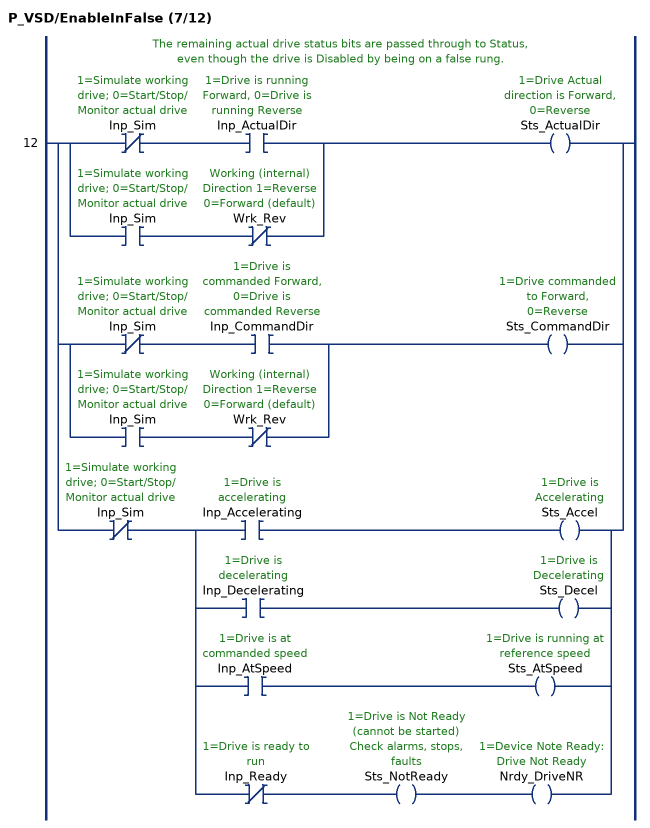
   // The remaining actual drive status bits are passed through to Status,
   // even though the drive is Disabled by being on a false rung.
   12: [[XIO(Inp_Sim) XIC(Inp_ActualDir) ,XIC(Inp_Sim) XIO(Wrk_Rev) ] OTE(Sts_ActualDir) ,[XIO(Inp_Sim) XIC(Inp_CommandDir) ,XIC(Inp_Sim) XIO(Wrk_Rev) ] OTE(Sts_CommandDir) ,XIO(Inp_Sim) [XIC(Inp_Accelerating) OTE(Sts_Accel) ,XIC(Inp_Decelerating) OTE(Sts_Decel) ,XIC(Inp_AtSpeed) OTE(Sts_AtSpeed) ,XIO(Inp_Ready) OTE(Sts_NotReady) OTE(Nrdy_DriveNR) ] ];
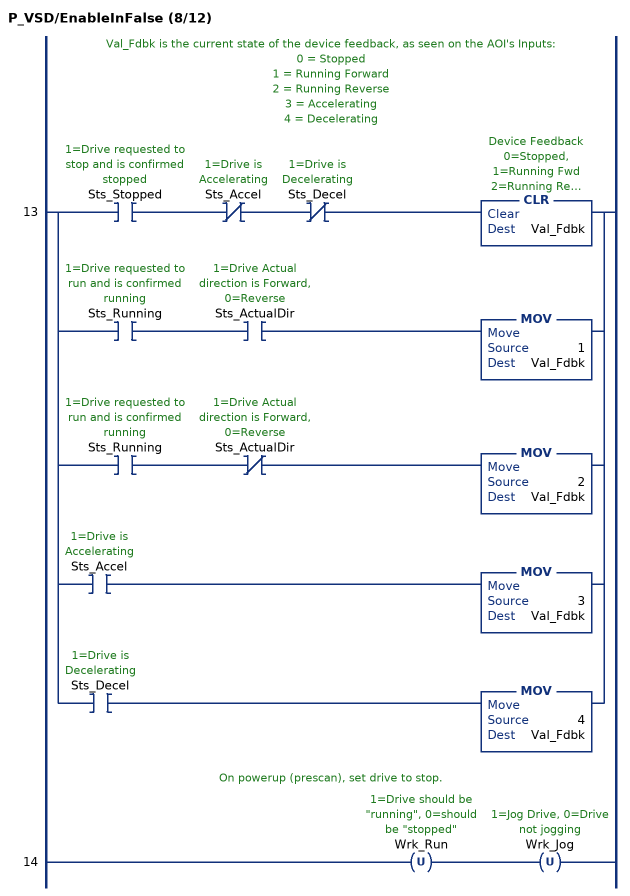
   // Val_Fdbk is the current state of the device feedback, as seen on the AOI's Inputs:
   // 0 = Stopped
   // 1 = Running Forward
   // 2 = Running Reverse
   // 3 = Accelerating
   // 4 = Decelerating
   13: [XIC(Sts_Stopped) XIO(Sts_Accel) XIO(Sts_Decel) CLR(Val_Fdbk) ,XIC(Sts_Running) XIC(Sts_ActualDir) MOV(1,Val_Fdbk) ,XIC(Sts_Running) XIO(Sts_ActualDir) MOV(2,Val_Fdbk) ,XIC(Sts_Accel) MOV(3,Val_Fdbk) ,XIC(Sts_Decel) MOV(4,Val_Fdbk) ];
   // On powerup (prescan), set drive to stop.
   14: OTU(Wrk_Run)OTU(Wrk_Jog);
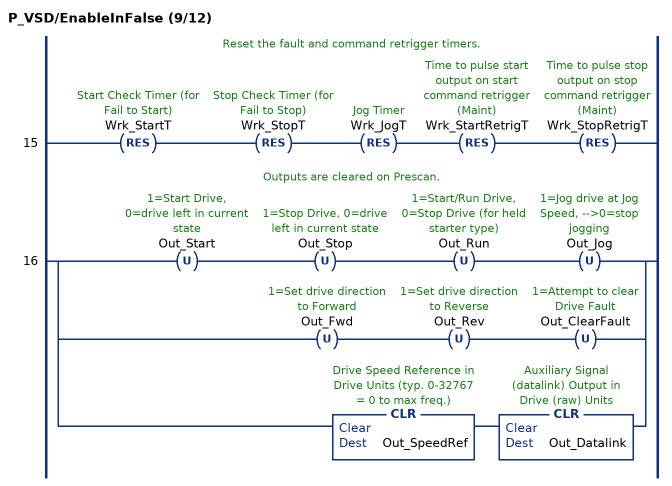
   // Reset the fault and command retrigger timers.
   15: RES(Wrk_StartT)RES(Wrk_StopT)RES(Wrk_JogT)RES(Wrk_StartRetrigT)RES(Wrk_StopRetrigT);
   // Outputs are cleared on Prescan.
   16: [OTU(Out_Start) OTU(Out_Stop) OTU(Out_Run) OTU(Out_Jog) ,OTU(Out_Fwd) OTU(Out_Rev) OTU(Out_ClearFault) ,CLR(Out_SpeedRef) CLR(Out_Datalink) ];
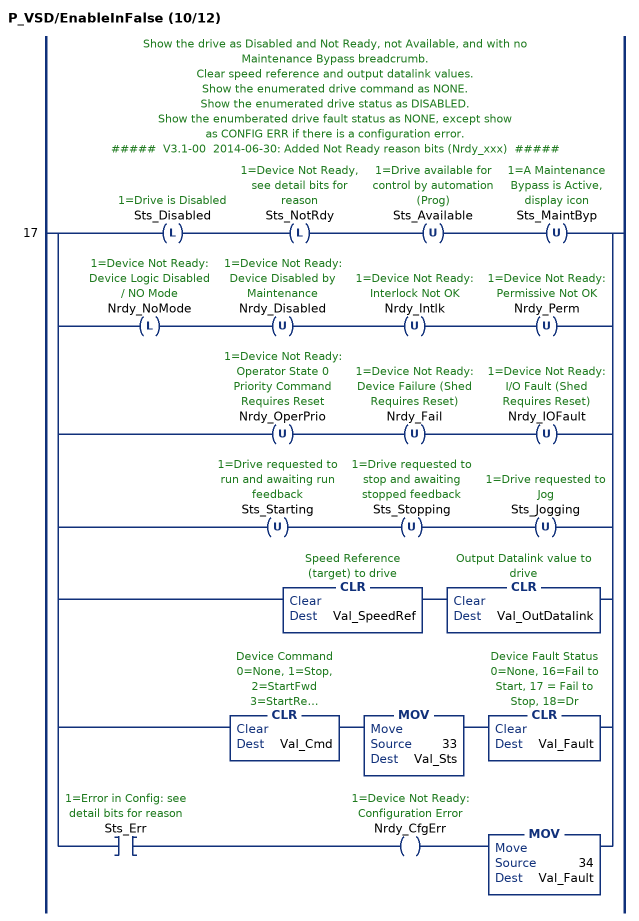
   // Show the drive as Disabled and Not Ready, not Available, and with no
   // Maintenance Bypass breadcrumb.
   // Clear speed reference and output datalink values.
   // Show the enumerated drive command as NONE.
   // Show the enumerated drive status as DISABLED.
   // Show the enumberated drive fault status as NONE, except show
   // as CONFIG ERR if there is a configuration error.
   // #####  V3.1-00  2014-06-30: Added Not Ready reason bits (Nrdy_xxx)  #####
   17: [OTL(Sts_Disabled) OTL(Sts_NotRdy) OTU(Sts_Available) OTU(Sts_MaintByp) ,OTL(Nrdy_NoMode) OTU(Nrdy_Disabled) OTU(Nrdy_Intlk) OTU(Nrdy_Perm) ,OTU(Nrdy_OperPrio) OTU(Nrdy_Fail) OTU(Nrdy_IOFault) ,OTU(Sts_Starting) OTU(Sts_Stopping) OTU(Sts_Jogging) ,CLR(Val_SpeedRef) CLR(Val_OutDatalink) ,CLR(Val_Cmd) MOV(33,Val_Sts) CLR(Val_Fault) ,XIC(Sts_Err) OTE(Nrdy_CfgErr) MOV(34,Val_Fault) ];
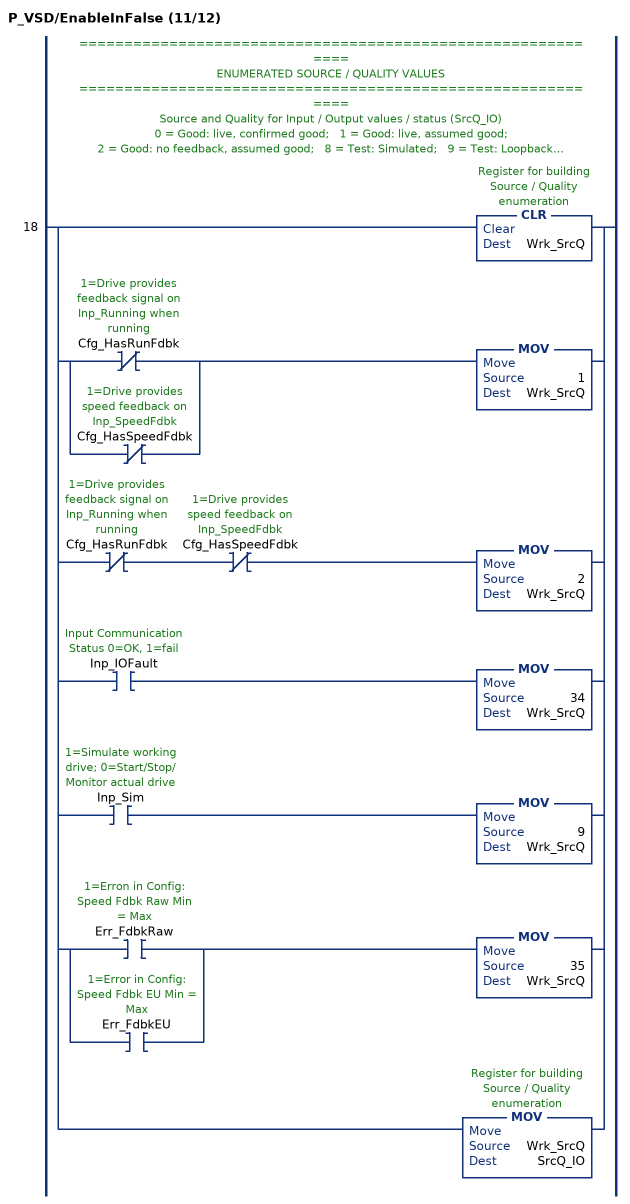
   // ============================================================
   // ENUMERATED SOURCE / QUALITY VALUES
   // ============================================================
   // Source and Quality for Input / Output values / status (SrcQ_IO)
   // 0 = Good: live, confirmed good;   1 = Good: live, assumed good;
   // 2 = Good: no feedback, assumed good;   8 = Test: Simulated;   9 = Test: Loopback;
   // 10 = Test: Manually Entered;   16 = Uncertain: Live, off-spec;
   // 17 = Uncertain, Substituted at Device / Bus;   18 = Uncertain, Substituted at AOI;
   // 19 = Uncertain, using last known good;    20 = Uncertain, using replacement value;
   // 32 = Bad, Signal Failure;   33 = Bad, Channel Fault;
   // 34 = Bad, Module / Comms Fault;   35 = Bad, Invalid Configuration
   // #####  V3.1-00  2014-06-30:  Added rung for Source/Quality enumerations.  #####
   18: [CLR(Wrk_SrcQ) ,[XIO(Cfg_HasRunFdbk) ,XIO(Cfg_HasSpeedFdbk) ] MOV(1,Wrk_SrcQ) ,XIO(Cfg_HasRunFdbk) XIO(Cfg_HasSpeedFdbk) MOV(2,Wrk_SrcQ) ,XIC(Inp_IOFault) MOV(34,Wrk_SrcQ) ,XIC(Inp_Sim) MOV(9,Wrk_SrcQ) ,[XIC(Err_FdbkRaw) ,XIC(Err_FdbkEU) ] MOV(35,Wrk_SrcQ) ,MOV(Wrk_SrcQ,SrcQ_IO) ];
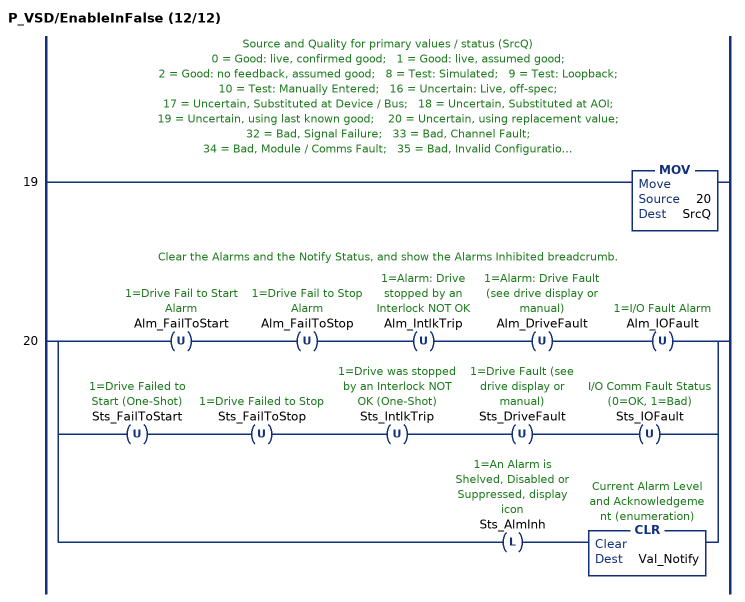
   // Source and Quality for primary values / status (SrcQ)
   // 0 = Good: live, confirmed good;   1 = Good: live, assumed good;
   // 2 = Good: no feedback, assumed good;   8 = Test: Simulated;   9 = Test: Loopback;
   // 10 = Test: Manually Entered;   16 = Uncertain: Live, off-spec;
   // 17 = Uncertain, Substituted at Device / Bus;   18 = Uncertain, Substituted at AOI;
   // 19 = Uncertain, using last known good;    20 = Uncertain, using replacement value;
   // 32 = Bad, Signal Failure;   33 = Bad, Channel Fault;
   // 34 = Bad, Module / Comms Fault;   35 = Bad, Invalid Configuration
   // #####  V3.1-00  2014-06-30:  Added rung for Source/Quality enumerations.  #####
   19: MOV(20,SrcQ);
   // Clear the Alarms and the Notify Status, and show the Alarms Inhibited breadcrumb.
   20: [OTU(Alm_FailToStart) OTU(Alm_FailToStop) OTU(Alm_IntlkTrip) OTU(Alm_DriveFault) OTU(Alm_IOFault) ,OTU(Sts_FailToStart) OTU(Sts_FailToStop) OTU(Sts_IntlkTrip) OTU(Sts_DriveFault) OTU(Sts_IOFault) ,OTL(Sts_AlmInh) CLR(Val_Notify) ];
END_ROUTINE

ROUTINE Logic   (* ladder *)
// Normal Scan: control / monitor Variable-Speed Drive
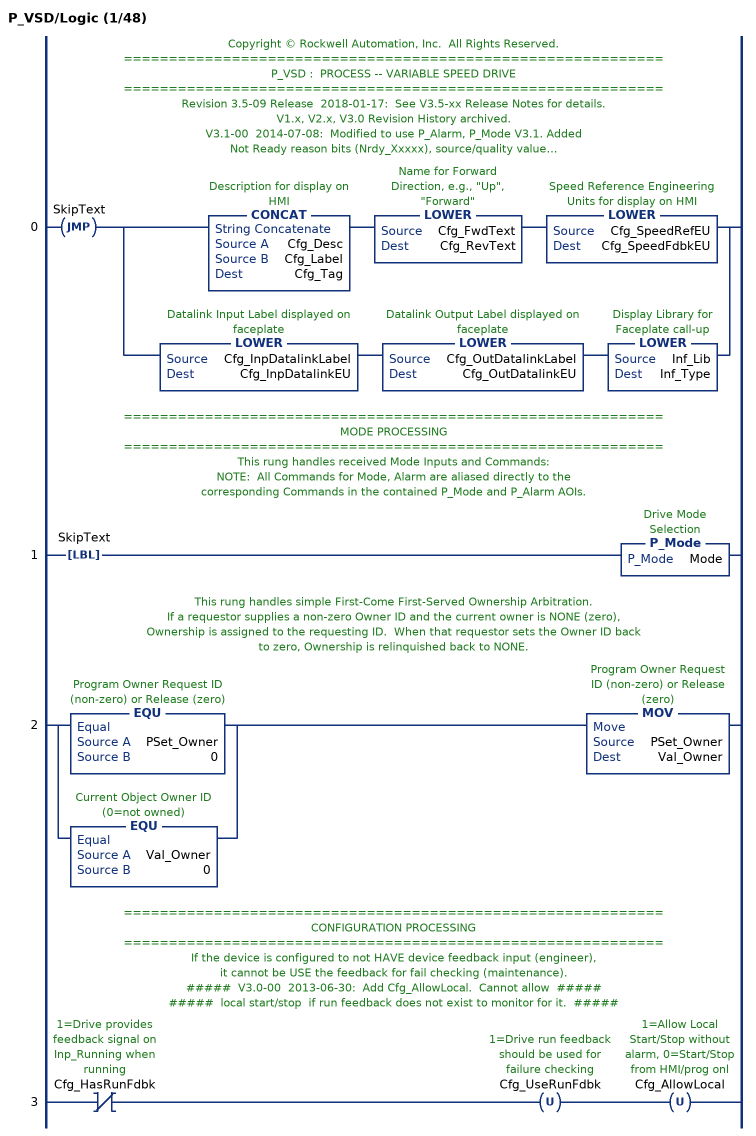
   // Copyright © Rockwell Automation, Inc.  All Rights Reserved.
   // ============================================================
   // P_VSD :  PROCESS -- VARIABLE SPEED DRIVE
   // ============================================================
   // Revision 3.5-09 Release  2018-01-17:  See V3.5-xx Release Notes for details.
   // V1.x, V2.x, V3.0 Revision History archived.
   // V3.1-00  2014-07-08:  Modified to use P_Alarm, P_Mode V3.1. Added
   // Not Ready reason bits (Nrdy_Xxxxx), source/quality values
   // (SrcQ). Modified default Parameter values
   // V3.1-01  2014-09-03:  Exposed jog, faill timers ACC/PRE (read-only). Corrections
   // to Nrdy_ trip and reset logic. Using P_Alarm, P_Mode V3.1-01.
   // V3.1-02  2014-09-30:  Unchanged, but using P_Alarm V3.1-02.
   // V3.1-03  2015-01-16;  Modified stop retriggering to handle asynchronous Prog mode owner.
   // V3.1-04 Patch01  2015-09-25:  Modified Val_SpeedFdbk generation when Cfg_HasSpeedFdbk = 0.
   // Changed description, use of Cfg_UseSpeedFdbk.
   // Modified to correct issue with loss of run feedback.
   // V3.1-05  2016-01-22:  Added Prescan check for OperKeep and ProgKeep both set.
   // V3.5-01  2016-01-29:  Unchanged, but using P_Alarm V3.5-01.
   // V3.5-02  2016-03-22:  Modified to eliminate oscillating Out_Stop on Drive Not Ready.
   // V3.5-04  2016-09-30:  Modified to handle Jog vs. Local Control; modified to align
   // with actual device state on transition from Sim to real drive.
   // V3.5-09  2018-01-17:  Modified to correct indication of motor RUNNING status in HAND
   // mode, regardless of interlock/stop conditions.
   // ============================================================
   // This Instruction controls and monitors a Variable-Speed Drive (AC or DC) and provides:
   // *  Starting, stopping, jogging of drive, setting speed reference and direction
   // *  Monitoring of run feedback, display of actual drive status, including accel, decel, direction, speed
   // *  Detection of Failure to Start, Failure to Stop, Drive Fault
   // *  Monitoring of Permissive conditions to allow starting
   // * Monitoring of Interlock conditions to stop / prevent starting
   // * Simulation, providing feedback of a working drive while disabling outputs
   // * Monitoring of I/O communication faults
   // * Alarms for Fail to Start, Fail to Stop, Interlock Trip, Drive Fault, I/O Fault
   // * Option to automatically reset faults and alarms when operator commands
   // motor to start or stop
   // * Supports HMI "breadcrumbs" for Alarm Inhibited, Bad Configuration,
   // Not Ready, Maintenance Bypass Active
   // * "Available" status for use by automation logic to know whether motor
   // can be controlled by other objects.
   // Modes are provided by a P_Mode Add-On Instruction instance.
   // Alarms are provided by P_Alarm Add-On Instruction instances.
   // Modes of operation: Operator, Program, Override, Maintenance, Hand
   // ============================================================
   // SHOW LOCAL STRINGS
   // ============================================================
   // The STRINGs containing the text associated with each instance of this
   // instruction cannot be Input or Output Parameters, because STRINGs are not
   //  'atomic' types. (Inputs and Outputs must be SINT, INT, DINT, REAL, or BOOL.)
   // In order to make it easier to find and configure these STRINGs, this rung
   // was added.  THE JMP (and the LBL on the following rung)
   // MUST NOT BE REMOVED!!!
   // To view the STRINGs, go to the instruction instance (in LD or FBD), RIGHT-click
   // to bring up the context menu and select "Open Instruction Logic".
   // This rung will appear with the STRING values for the selected instance.
   // You may double-click the STRING values here to modify them as well.
   // #####  V3.0-00  2013-06-30:  Added Val_FaultDesc to strings shown by this rung.  #####
   0: JMP(SkipText)[CONCAT(Cfg_Desc,Cfg_Label,Cfg_Tag) LOWER(Cfg_FwdText,Cfg_RevText) LOWER(Cfg_SpeedRefEU,Cfg_SpeedFdbkEU) ,LOWER(Cfg_InpDatalinkLabel,Cfg_InpDatalinkEU) LOWER(Cfg_OutDatalinkLabel,Cfg_OutDatalinkEU) LOWER(Inf_Lib,Inf_Type) ];
   // ============================================================
   // MODE PROCESSING
   // ============================================================
   // This rung handles received Mode Inputs and Commands:
   // NOTE:  All Commands for Mode, Alarm are aliased directly to the
   // corresponding Commands in the contained P_Mode and P_Alarm AOIs.
   1: LBL(SkipText)P_Mode(Mode);
   // This rung handles simple First-Come First-Served Ownership Arbitration.
   // If a requestor supplies a non-zero Owner ID and the current owner is NONE (zero),
   // Ownership is assigned to the requesting ID.  When that requestor sets the Owner ID back
   // to zero, Ownership is relinquished back to NONE.
   2: [EQU(PSet_Owner,0) ,EQU(Val_Owner,0) ]MOV(PSet_Owner,Val_Owner);
   // ============================================================
   // CONFIGURATION PROCESSING
   // ============================================================
   // If the device is configured to not HAVE device feedback input (engineer),
   // it cannot be USE the feedback for fail checking (maintenance).
   // #####  V3.0-00  2013-06-30:  Add Cfg_AllowLocal.  Cannot allow  #####
   // #####  local start/stop  if run feedback does not exist to monitor for it.  #####
   3: XIO(Cfg_HasRunFdbk)OTU(Cfg_UseRunFdbk)OTU(Cfg_AllowLocal);
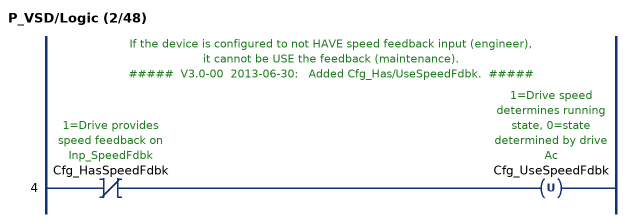
   // If the device is configured to not HAVE speed feedback input (engineer),
   // it cannot be USE the feedback (maintenance).
   // #####  V3.0-00  2013-06-30:   Added Cfg_Has/UseSpeedFdbk.  #####
   4: XIO(Cfg_HasSpeedFdbk)OTU(Cfg_UseSpeedFdbk);
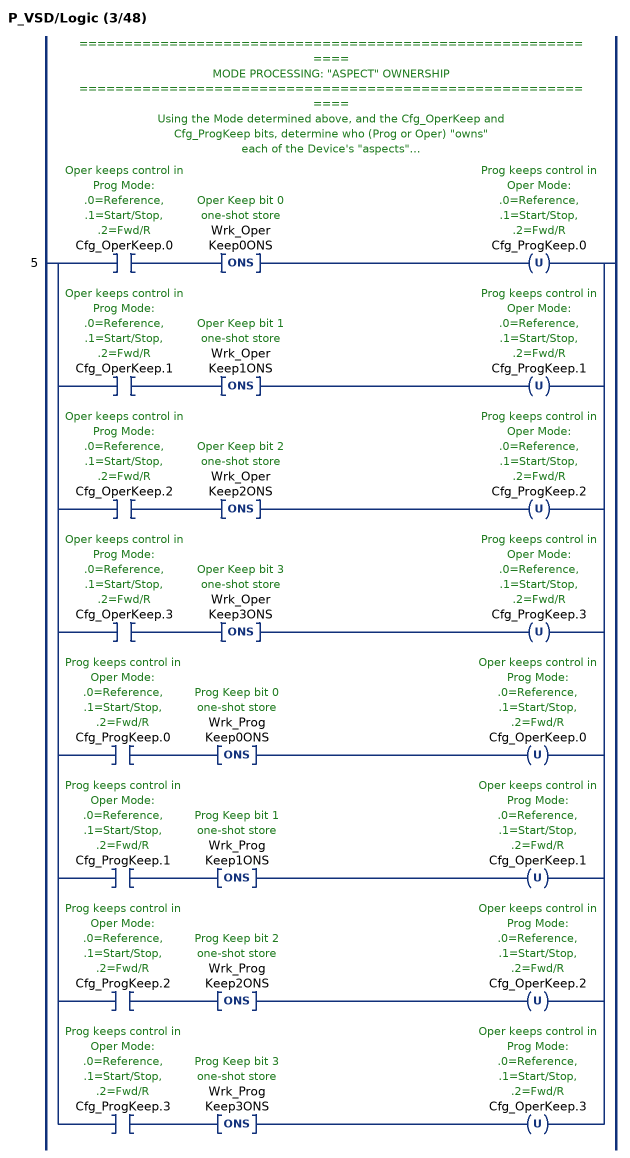
   // ============================================================
   // MODE PROCESSING: "ASPECT" OWNERSHIP
   // ============================================================
   // Using the Mode determined above, and the Cfg_OperKeep and
   // Cfg_ProgKeep bits, determine who (Prog or Oper) "owns"
   // each of the Device's "aspects":
   // Speed Reference (.0), Start/Stop (.1),
   // Forward/Reverse (.2), and Output Datalink (.3).
   // The bits within Cfg_OperKeep and Cfg_ProgKeep determine which "aspects"
   // (sub-functions of this AOI) are retained by the Operator in Program Mode,
   // or by the Program in Operator Mode (respectively).
   // All aspects (functions) may be "kept" (basically locking the Operator/Program Mode
   // selection, rendering it moot --  you get to explain how it works to your operators!!!),
   // but it is NOT allowed to have any given function retained by BOTH Operator and
   // Program.  This rung ensures that no function is "kept" by both Oper and Prog.
   5: [XIC(Cfg_OperKeep.0) ONS(Wrk_OperKeep0ONS) OTU(Cfg_ProgKeep.0) ,XIC(Cfg_OperKeep.1) ONS(Wrk_OperKeep1ONS) OTU(Cfg_ProgKeep.1) ,XIC(Cfg_OperKeep.2) ONS(Wrk_OperKeep2ONS) OTU(Cfg_ProgKeep.2) ,XIC(Cfg_OperKeep.3) ONS(Wrk_OperKeep3ONS) OTU(Cfg_ProgKeep.3) ,XIC(Cfg_ProgKeep.0) ONS(Wrk_ProgKeep0ONS) OTU(Cfg_OperKeep.0) ,XIC(Cfg_ProgKeep.1) ONS(Wrk_ProgKeep1ONS) OTU(Cfg_OperKeep.1) ,XIC(Cfg_ProgKeep.2) ONS(Wrk_ProgKeep2ONS) OTU(Cfg_OperKeep.2) ,XIC(Cfg_ProgKeep.3) ONS(Wrk_ProgKeep3ONS) OTU(Cfg_OperKeep.3) ];
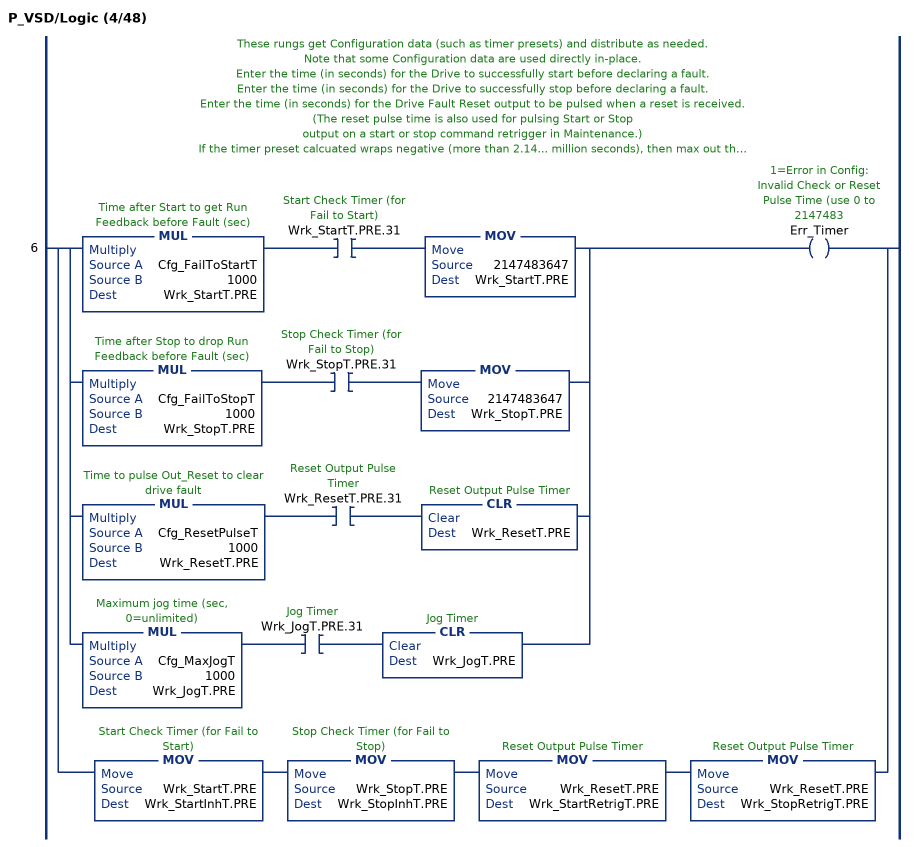
   // These rungs get Configuration data (such as timer presets) and distribute as needed.
   // Note that some Configuration data are used directly in-place.
   // Enter the time (in seconds) for the Drive to successfully start before declaring a fault.
   // Enter the time (in seconds) for the Drive to successfully stop before declaring a fault.
   // Enter the time (in seconds) for the Drive Fault Reset output to be pulsed when a reset is received.
   // (The reset pulse time is also used for pulsing Start or Stop
   // output on a start or stop command retrigger in Maintenance.)
   // If the timer preset calcuated wraps negative (more than 2.14... million seconds), then max out the
   // or clear the Timer Preset (as appropriate) and flag it.  Note that a negative timer preset will fault the controller!!!
   // #####  V3.1-04 Patch01  2015-09-25:  Modified to correct issue with loss of run feedback.  #####
   6: [[MUL(Cfg_FailToStartT,1000,Wrk_StartT.PRE) XIC(Wrk_StartT.PRE.31) MOV(2147483647,Wrk_StartT.PRE) ,MUL(Cfg_FailToStopT,1000,Wrk_StopT.PRE) XIC(Wrk_StopT.PRE.31) MOV(2147483647,Wrk_StopT.PRE) ,MUL(Cfg_ResetPulseT,1000,Wrk_ResetT.PRE) XIC(Wrk_ResetT.PRE.31) CLR(Wrk_ResetT.PRE) ,MUL(Cfg_MaxJogT,1000,Wrk_JogT.PRE) XIC(Wrk_JogT.PRE.31) CLR(Wrk_JogT.PRE) ] OTE(Err_Timer) ,MOV(Wrk_StartT.PRE,Wrk_StartInhT.PRE) MOV(Wrk_StopT.PRE,Wrk_StopInhT.PRE) MOV(Wrk_ResetT.PRE,Wrk_StartRetrigT.PRE) MOV(Wrk_ResetT.PRE,Wrk_StopRetrigT.PRE) ];
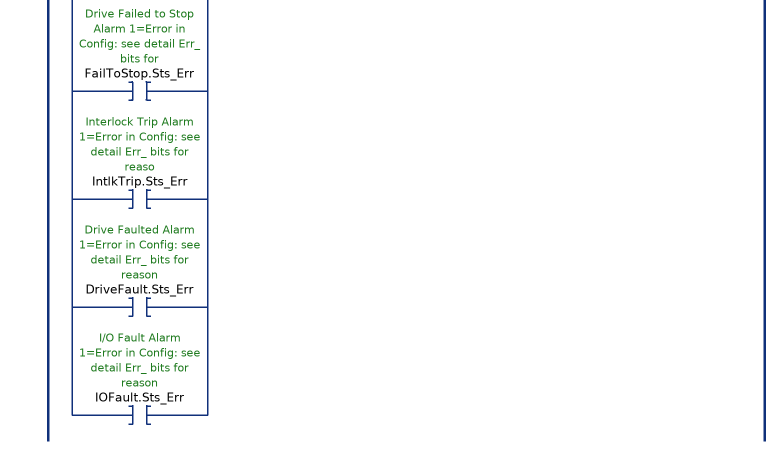
   // This rung handles the reports of all Bad Configuration Status.
   // Individual bits are provided for various status:
   // Bad Raw Scaling configs
   // Bad Engineering Units Scaling configs
   // Bad Min or Max Speed Reference clamp limit
   // Bad simulation speed ramp time
   // Bad timer config from (rung above)
   // Bad Alarm config (from P_Alarm)
   // Bad Cfg_OperKeep / Cfg_ProgKeep config
   // Then a summary Bad Config status is provided, simply an OR of the individual bits.
   // #####  V3.0-00  2013-06-30:   Added Cfg_HasSpeedFdbk  #####
   7: [XIC(Cfg_HasSpeedFdbk) [EQU(Cfg_SpeedFdbkRawMax,Cfg_SpeedFdbkRawMin) OTE(Err_FdbkRaw) ,EQU(Cfg_SpeedFdbkEUMax,Cfg_SpeedFdbkEUMin) OTE(Err_FdbkEU) ] ,EQU(Cfg_SpeedRefEUMax,Cfg_SpeedRefEUMin) OTE(Err_RefEU) ,EQU(Cfg_SpeedRefRawMax,Cfg_SpeedRefRawMin) OTE(Err_RefRaw) ,XIC(Cfg_HasInpDatalink) [EQU(Cfg_InpDatalinkRawMax,Cfg_InpDatalinkRawMin) OTE(Err_InpDLRaw) ,EQU(Cfg_InpDatalinkEUMax,Cfg_InpDatalinkEUMin) OTE(Err_InpDLEU) ] ,XIC(Cfg_HasOutDatalink) [LEQ(Cfg_OutDatalinkMax,Cfg_OutDatalinkMin) OTE(Err_OutDLLim) ,EQU(Cfg_OutDatalinkEUMax,Cfg_OutDatalinkEUMin) OTE(Err_OutDLEU) ,EQU(Cfg_OutDatalinkRawMax,Cfg_OutDatalinkRawMin) OTE(Err_OutDLRaw) ] ,[LEQ(Cfg_MaxSpdRef,Cfg_MinSpdRef) ,LES(Cfg_MinSpdRef,0.0) ] OTE(Err_RefLim) ,LES(Cfg_SimRampT,0) OTE(Err_Sim) ,XIC(Err_Timer) ,[XIC(FailToStart.Sts_Err) ,XIC(FailToStop.Sts_Err) ,XIC(IntlkTrip.Sts_Err) ,XIC(DriveFault.Sts_Err) ,XIC(IOFault.Sts_Err) ] OTE(Err_Alarm) ]OTE(Sts_Err);
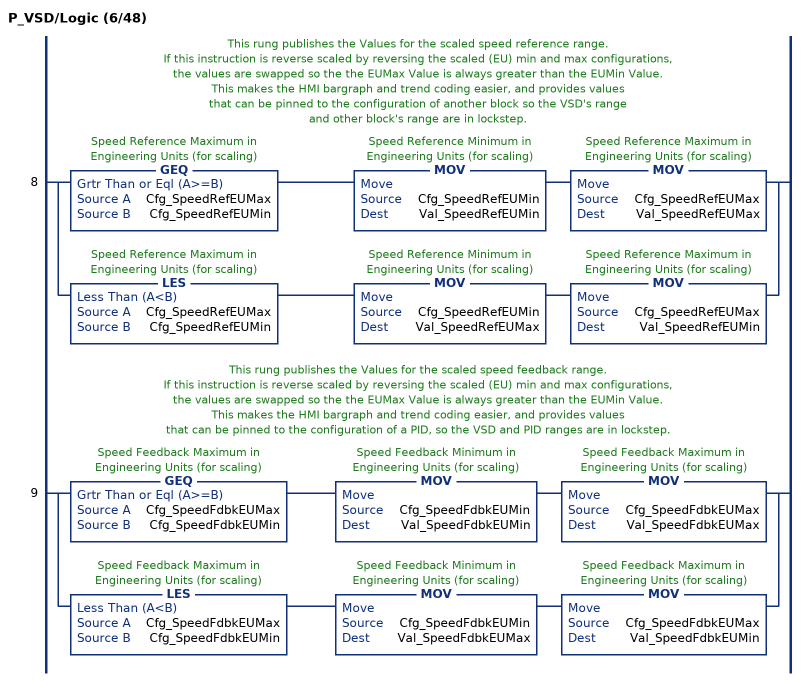
   // This rung publishes the Values for the scaled speed reference range.
   // If this instruction is reverse scaled by reversing the scaled (EU) min and max configurations,
   // the values are swapped so the the EUMax Value is always greater than the EUMin Value.
   // This makes the HMI bargraph and trend coding easier, and provides values
   // that can be pinned to the configuration of another block so the VSD's range
   //  and other block's range are in lockstep.
   8: [GEQ(Cfg_SpeedRefEUMax,Cfg_SpeedRefEUMin) MOV(Cfg_SpeedRefEUMin,Val_SpeedRefEUMin) MOV(Cfg_SpeedRefEUMax,Val_SpeedRefEUMax) ,LES(Cfg_SpeedRefEUMax,Cfg_SpeedRefEUMin) MOV(Cfg_SpeedRefEUMin,Val_SpeedRefEUMax) MOV(Cfg_SpeedRefEUMax,Val_SpeedRefEUMin) ];
   // This rung publishes the Values for the scaled speed feedback range.
   // If this instruction is reverse scaled by reversing the scaled (EU) min and max configurations,
   // the values are swapped so the the EUMax Value is always greater than the EUMin Value.
   // This makes the HMI bargraph and trend coding easier, and provides values
   // that can be pinned to the configuration of a PID, so the VSD and PID ranges are in lockstep.
   9: [GEQ(Cfg_SpeedFdbkEUMax,Cfg_SpeedFdbkEUMin) MOV(Cfg_SpeedFdbkEUMin,Val_SpeedFdbkEUMin) MOV(Cfg_SpeedFdbkEUMax,Val_SpeedFdbkEUMax) ,LES(Cfg_SpeedFdbkEUMax,Cfg_SpeedFdbkEUMin) MOV(Cfg_SpeedFdbkEUMin,Val_SpeedFdbkEUMax) MOV(Cfg_SpeedFdbkEUMax,Val_SpeedFdbkEUMin) ];
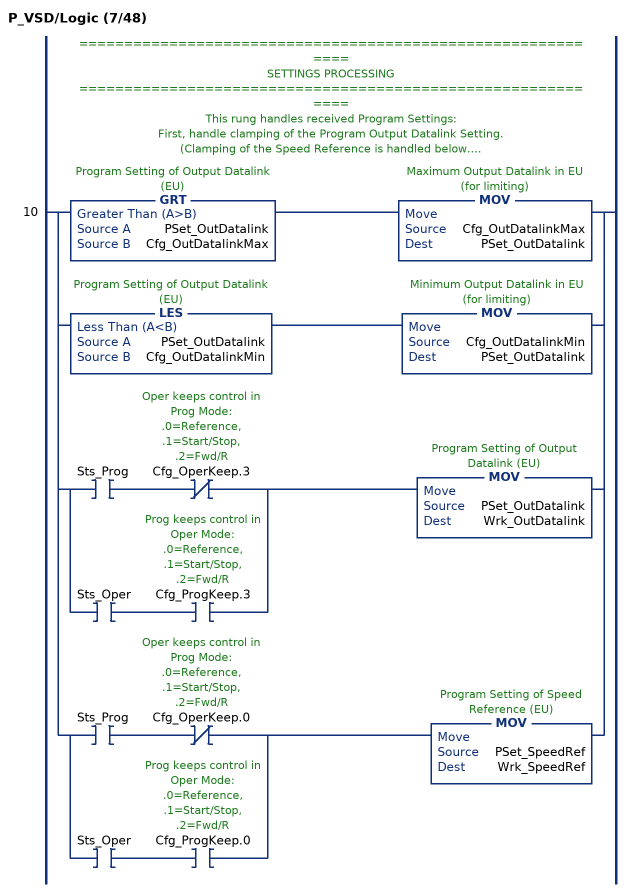
   // ============================================================
   // SETTINGS PROCESSING
   // ============================================================
   // This rung handles received Program Settings:
   // First, handle clamping of the Program Output Datalink Setting.
   // (Clamping of the Speed Reference is handled below.)
   // Then, if the Mode is Program and the Operator does not retain the Output Datalink,
   // or if the Mode is Operator but the Program retains the Output Datalink,
   // use the Program Setting for the Output Datalink.
   // The Program Setting for the Speed Reference is handled similarly.
   10: [GRT(PSet_OutDatalink,Cfg_OutDatalinkMax) MOV(Cfg_OutDatalinkMax,PSet_OutDatalink) ,LES(PSet_OutDatalink,Cfg_OutDatalinkMin) MOV(Cfg_OutDatalinkMin,PSet_OutDatalink) ,[XIC(Sts_Prog) XIO(Cfg_OperKeep.3) ,XIC(Sts_Oper) XIC(Cfg_ProgKeep.3) ] MOV(PSet_OutDatalink,Wrk_OutDatalink) ,[XIC(Sts_Prog) XIO(Cfg_OperKeep.0) ,XIC(Sts_Oper) XIC(Cfg_ProgKeep.0) ] MOV(PSet_SpeedRef,Wrk_SpeedRef) ];
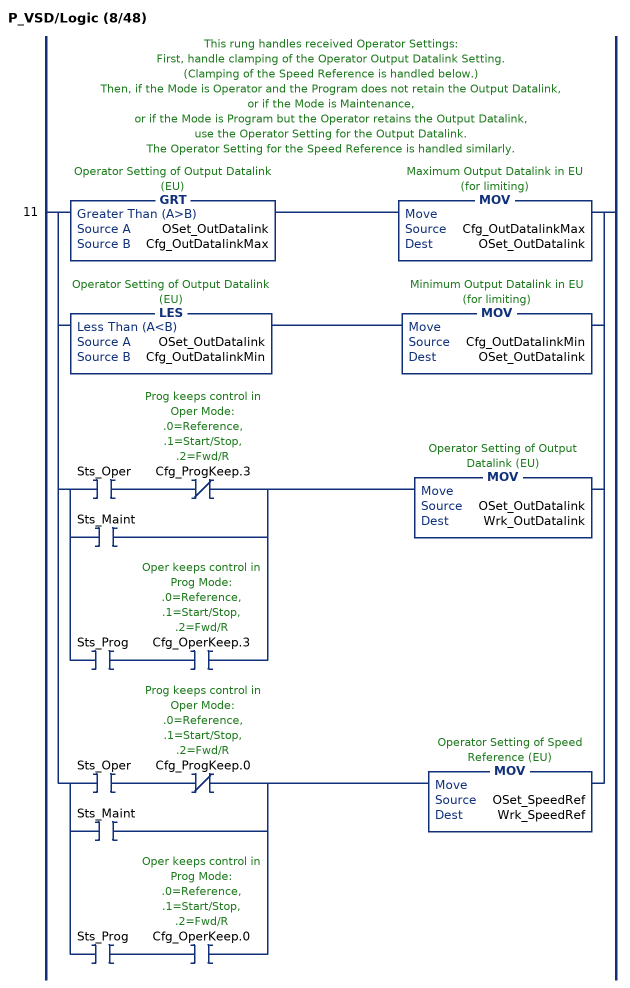
   // This rung handles received Operator Settings:
   // First, handle clamping of the Operator Output Datalink Setting.
   // (Clamping of the Speed Reference is handled below.)
   // Then, if the Mode is Operator and the Program does not retain the Output Datalink,
   // or if the Mode is Maintenance,
   // or if the Mode is Program but the Operator retains the Output Datalink,
   // use the Operator Setting for the Output Datalink.
   // The Operator Setting for the Speed Reference is handled similarly.
   11: [GRT(OSet_OutDatalink,Cfg_OutDatalinkMax) MOV(Cfg_OutDatalinkMax,OSet_OutDatalink) ,LES(OSet_OutDatalink,Cfg_OutDatalinkMin) MOV(Cfg_OutDatalinkMin,OSet_OutDatalink) ,[XIC(Sts_Oper) XIO(Cfg_ProgKeep.3) ,XIC(Sts_Maint) ,XIC(Sts_Prog) XIC(Cfg_OperKeep.3) ] MOV(OSet_OutDatalink,Wrk_OutDatalink) ,[XIC(Sts_Oper) XIO(Cfg_ProgKeep.0) ,XIC(Sts_Maint) ,XIC(Sts_Prog) XIC(Cfg_OperKeep.0) ] MOV(OSet_SpeedRef,Wrk_SpeedRef) ];
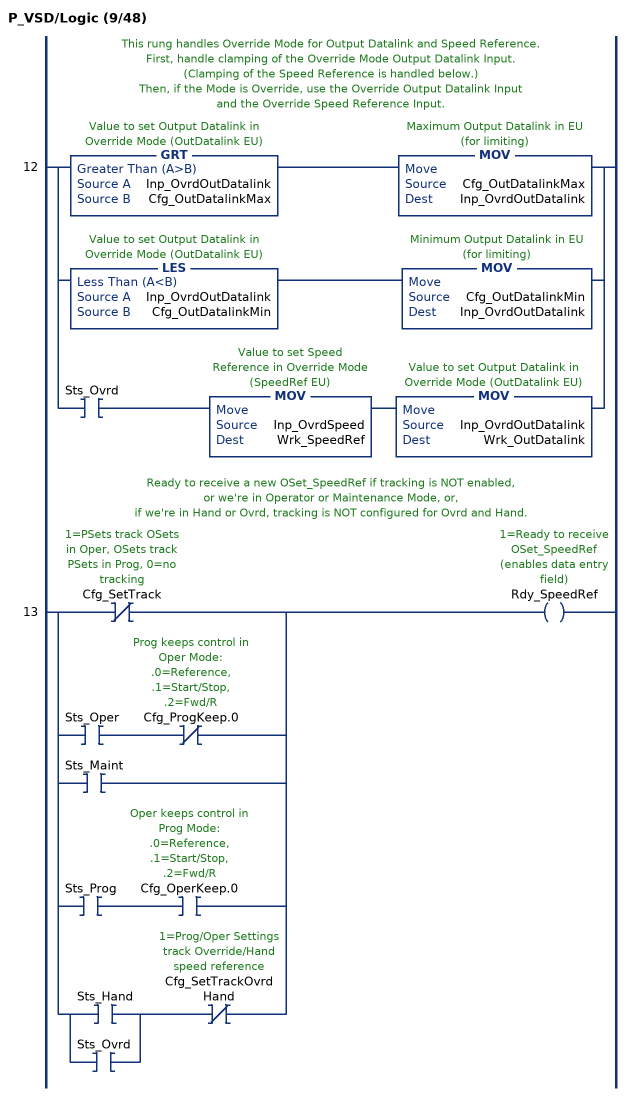
   // This rung handles Override Mode for Output Datalink and Speed Reference.
   // First, handle clamping of the Override Mode Output Datalink Input.
   // (Clamping of the Speed Reference is handled below.)
   // Then, if the Mode is Override, use the Override Output Datalink Input
   // and the Override Speed Reference Input.
   12: [GRT(Inp_OvrdOutDatalink,Cfg_OutDatalinkMax) MOV(Cfg_OutDatalinkMax,Inp_OvrdOutDatalink) ,LES(Inp_OvrdOutDatalink,Cfg_OutDatalinkMin) MOV(Cfg_OutDatalinkMin,Inp_OvrdOutDatalink) ,XIC(Sts_Ovrd) MOV(Inp_OvrdSpeed,Wrk_SpeedRef) MOV(Inp_OvrdOutDatalink,Wrk_OutDatalink) ];
   // Ready to receive a new OSet_SpeedRef if tracking is NOT enabled,
   // or we're in Operator or Maintenance Mode, or,
   // if we're in Hand or Ovrd, tracking is NOT configured for Ovrd and Hand.
   13: [XIO(Cfg_SetTrack) ,XIC(Sts_Oper) XIO(Cfg_ProgKeep.0) ,XIC(Sts_Maint) ,XIC(Sts_Prog) XIC(Cfg_OperKeep.0) ,[XIC(Sts_Hand) ,XIC(Sts_Ovrd) ] XIO(Cfg_SetTrackOvrdHand) ]OTE(Rdy_SpeedRef);
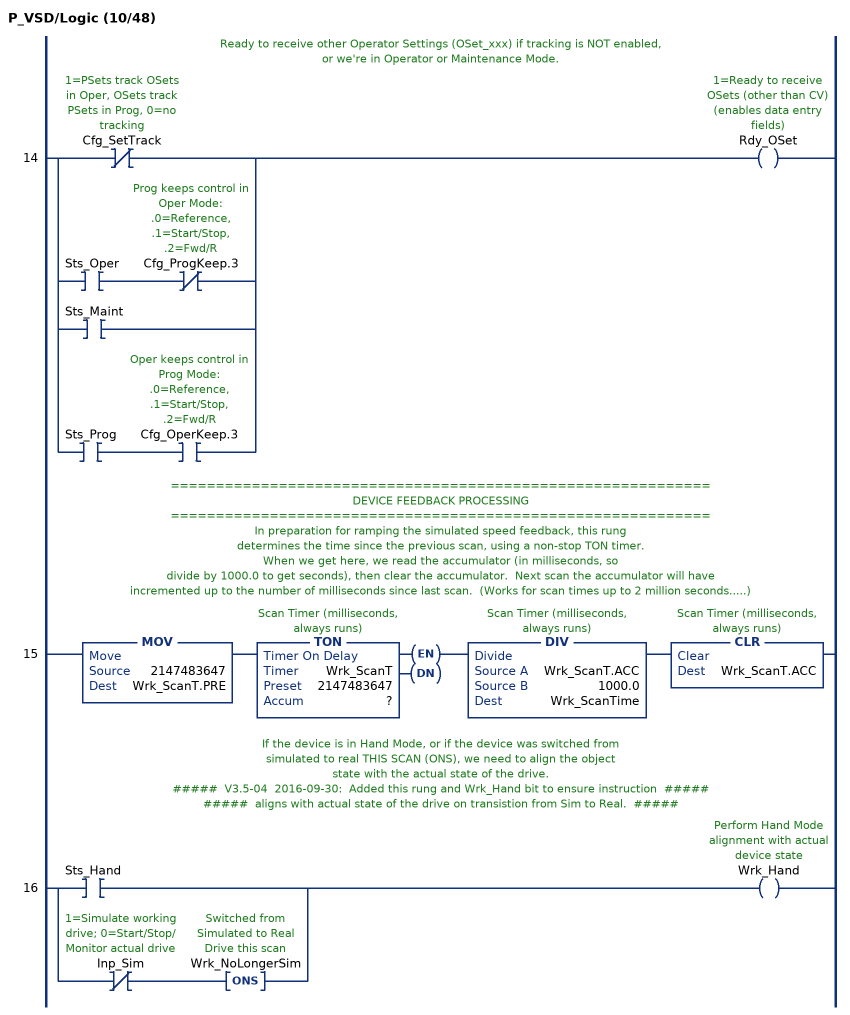
   // Ready to receive other Operator Settings (OSet_xxx) if tracking is NOT enabled,
   // or we're in Operator or Maintenance Mode.
   14: [XIO(Cfg_SetTrack) ,XIC(Sts_Oper) XIO(Cfg_ProgKeep.3) ,XIC(Sts_Maint) ,XIC(Sts_Prog) XIC(Cfg_OperKeep.3) ]OTE(Rdy_OSet);
   // ============================================================
   // DEVICE FEEDBACK PROCESSING
   // ============================================================
   // In preparation for ramping the simulated speed feedback, this rung
   // determines the time since the previous scan, using a non-stop TON timer.
   // When we get here, we read the accumulator (in milliseconds, so
   // divide by 1000.0 to get seconds), then clear the accumulator.  Next scan the accumulator will have
   // incremented up to the number of milliseconds since last scan.  (Works for scan times up to 2 million seconds.....)
   15: MOV(2147483647,Wrk_ScanT.PRE)TON(Wrk_ScanT,?,?)DIV(Wrk_ScanT.ACC,1000.0,Wrk_ScanTime)CLR(Wrk_ScanT.ACC);
   // If the device is in Hand Mode, or if the device was switched from
   // simulated to real THIS SCAN (ONS), we need to align the object
   // state with the actual state of the drive.
   // #####  V3.5-04  2016-09-30:  Added this rung and Wrk_Hand bit to ensure instruction  #####
   // #####  aligns with actual state of the drive on transistion from Sim to Real.  #####
   16: [XIC(Sts_Hand) ,XIO(Inp_Sim) ONS(Wrk_NoLongerSim) ]OTE(Wrk_Hand);
